(* PLC project mtcs_axes, Institute of Astronomy Onto 0.0.1 *)
(* stored: creationDateTime 2025-02-15T22:09:55.843531, modificationDateTime 2025-02-15T22:09:55.843531 *)

TYPE AxesIds : (AZI := 0, ABL := 1, ELE := 2, ROC := 3, RON := 4);
END_TYPE

TYPE AxesMoveUnits : (DEGREES := 0, RADIANS := 1, ARCSECONDS := 2);
END_TYPE

TYPE AxesAlphaUnits : (HOURS := 0, DEGREES := 1, RADIANS := 2);
END_TYPE

TYPE AxesDeltaUnits : (DEGREES := 0, RADIANS := 1);
END_TYPE

TYPE AxesMuUnits : (ARCSECONDS_PER_YEAR := 0, MILLIARCSECONDS_PER_YEAR := 1, DEGREES_PER_YEAR := 2, RADIANS_PER_YEAR := 3);
END_TYPE

TYPE AxesMoveVelocityUnits : (DEGREES_PER_SECOND := 0, ARCSECONDS_PER_SECOND := 1, RADIANS_PER_SECOND := 2, ARCSECONDS_PER_MINUTE := 3, ARCSECONDS_PER_HOUR := 4);
END_TYPE

TYPE AxesRotatorActivity : (NONE_ACTIVE := 0, ROC_ACTIVE := 1, RON_ACTIVE := 2);
END_TYPE

TYPE AxesParts : STRUCT
  {attribute 'TcHmiSymbol.Show'}
  azi : AxesAzimuthAxis;  (* The azimuth axis *)
  {attribute 'TcHmiSymbol.Show'}
  ele : AxesElevationAxis;  (* The elevation axis *)
  {attribute 'TcHmiSymbol.Show'}
  roc : AxesRotationAxis;  (* The cassegrain derotator axis *)
  {attribute 'TcHmiSymbol.Show'}
  ron : AxesRotationAxis;  (* The nasmyth derotator axis *)
  {attribute 'TcHmiSymbol.Show'}
  io : AxesIO;  (* I/O modules and drives *)
  {attribute 'TcHmiSymbol.Show'}
  configManager : ConfigManager;  (* The config manager (to load/save/activate configuration data) *)
  {attribute 'TcHmiSymbol.Show'}
  tpoint : AxesPointingModelsSetup;  (* The TPOINT models setup *)
END_STRUCT;
END_TYPE

TYPE AxesAzimuthAxisParts : STRUCT
  {attribute 'TcHmiSymbol.Show'}
  virtualAxis : AngularAxis;  (* The virtual AZI axis *)
  {attribute 'TcHmiSymbol.Show'}
  physicalAxis : AngularAxis;  (* The physical AZI axis *)
  {attribute 'TcHmiSymbol.Show'}
  ablAxis : AngularAxis;  (* The (anti-backlash) ABL axis *)
  {attribute 'TcHmiSymbol.Show'}
  lida1 : IncrementalEncoder;  (* The external (LIDA) encoder no. 1 *)
  {attribute 'TcHmiSymbol.Show'}
  lida2 : IncrementalEncoder;  (* The external (LIDA) encoder no. 2 *)
  {attribute 'TcHmiSymbol.Show'}
  lida3 : IncrementalEncoder;  (* The external (LIDA) encoder no. 3 *)
  {attribute 'TcHmiSymbol.Show'}
  lida4 : IncrementalEncoder;  (* The external (LIDA) encoder no. 4 *)
  {attribute 'TcHmiSymbol.Show'}
  absoluteEncoder : SSIEncoder;  (* The external absolute encoder *)
END_STRUCT;
END_TYPE

TYPE AxesElevationAxisParts : STRUCT
  {attribute 'TcHmiSymbol.Show'}
  virtualAxis : AngularAxis;  (* The virtual axis *)
  {attribute 'TcHmiSymbol.Show'}
  physicalAxis : AngularAxis;  (* The physical ELE axis *)
  {attribute 'TcHmiSymbol.Show'}
  lida1 : IncrementalEncoder;  (* The external (LIDA) encoder no. 1 *)
  {attribute 'TcHmiSymbol.Show'}
  lida2 : IncrementalEncoder;  (* The external (LIDA) encoder no. 2 *)
  {attribute 'TcHmiSymbol.Show'}
  absoluteEncoder : SSIEncoder;  (* The external absolute encoder *)
END_STRUCT;
END_TYPE

TYPE AxesRotationAxisParts : STRUCT
  {attribute 'TcHmiSymbol.Show'}
  virtualAxis : AngularAxis;  (* The virtual axis *)
  {attribute 'TcHmiSymbol.Show'}
  physicalAxis : AngularAxis;  (* The physical axis *)
END_STRUCT;
END_TYPE

TYPE AxesPointingModelSetupParts : STRUCT
  {attribute 'TcHmiSymbol.Show'}
  configManager : ConfigManager;  (* The config manager (to load/save/activate configuration data) *)
END_STRUCT;
END_TYPE

TYPE AxesPointingModelsSetupParts : STRUCT
  {attribute 'TcHmiSymbol.Show'}
  model0 : AxesPointingModelSetup;
  {attribute 'TcHmiSymbol.Show'}
  model1 : AxesPointingModelSetup;
  {attribute 'TcHmiSymbol.Show'}
  model2 : AxesPointingModelSetup;
  {attribute 'TcHmiSymbol.Show'}
  model3 : AxesPointingModelSetup;
  {attribute 'TcHmiSymbol.Show'}
  model4 : AxesPointingModelSetup;
  {attribute 'TcHmiSymbol.Show'}
  model5 : AxesPointingModelSetup;
  {attribute 'TcHmiSymbol.Show'}
  model6 : AxesPointingModelSetup;
  {attribute 'TcHmiSymbol.Show'}
  model7 : AxesPointingModelSetup;
  {attribute 'TcHmiSymbol.Show'}
  model8 : AxesPointingModelSetup;
  {attribute 'TcHmiSymbol.Show'}
  model9 : AxesPointingModelSetup;
END_STRUCT;
END_TYPE

TYPE AxesIOParts : STRUCT
  {attribute 'TcHmiSymbol.Show'}
  aziDrive : AX52XXDrive;  (* The AX5000 drive for the AZI en ROC motors *)
  {attribute 'TcHmiSymbol.Show'}
  ablDrive : AX52XXDrive;  (* The AX5000 drive for the ABL en RON motors *)
  {attribute 'TcHmiSymbol.Show'}
  eleDrive : AX52XXDrive;  (* The AX5000 drive for the ELE en FW motors *)
  {attribute 'TcHmiSymbol.Show'}
  TA_AZID : EtherCatDevice;  (* Telescope Axis - AZID *)
  {attribute 'TcHmiSymbol.Show'}
  TA_ABLD : EtherCatDevice;  (* Telescope Axis - ABLD *)
  {attribute 'TcHmiSymbol.Show'}
  TA_ELED : EtherCatDevice;  (* Telescope Axis - ELED *)
  {attribute 'TcHmiSymbol.Show'}
  TE_COU : EtherCatDevice;  (* Telescope Encoders - COU *)
  {attribute 'TcHmiSymbol.Show'}
  TE_EN1 : EtherCatDevice;  (* Telescope Encoders - EN1 *)
  {attribute 'TcHmiSymbol.Show'}
  TE_EN2 : EtherCatDevice;  (* Telescope Encoders - EN2 *)
  {attribute 'TcHmiSymbol.Show'}
  TE_EN3 : EtherCatDevice;  (* Telescope Encoders - EN3 *)
  {attribute 'TcHmiSymbol.Show'}
  TE_EN4 : EtherCatDevice;  (* Telescope Encoders - EN4 *)
  {attribute 'TcHmiSymbol.Show'}
  TE_EN5 : EtherCatDevice;  (* Telescope Encoders - EN5 *)
  {attribute 'TcHmiSymbol.Show'}
  TE_EN6 : EtherCatDevice;  (* Telescope Encoders - EN6 *)
  {attribute 'TcHmiSymbol.Show'}
  TE_EN7 : EtherCatDevice;  (* Telescope Encoders - EN7 *)
END_STRUCT;
END_TYPE

TYPE AxesProcesses : STRUCT
  {attribute 'TcHmiSymbol.Show'}
  initialize : Process;  (* Start initializing *)
  {attribute 'TcHmiSymbol.Show'}
  reset : Process;  (* Reset the axis (no homing) *)
  {attribute 'TcHmiSymbol.Show'}
  lock : Process;  (* Lock the system *)
  {attribute 'TcHmiSymbol.Show'}
  unlock : Process;  (* Unlock the system *)
  {attribute 'TcHmiSymbol.Show'}
  changeOperatingState : ChangeOperatingStateProcess;  (* Change the operating state (e.g. AUTO, MANUAL, ...) *)
  {attribute 'TcHmiSymbol.Show'}
  setTarget : AxesSetTargetProcess;  (* Set a new target *)
  {attribute 'TcHmiSymbol.Show'}
  point : AxesPointProcess;  (* Point the telescope to a new target *)
  {attribute 'TcHmiSymbol.Show'}
  pointRelative : AxesPointRelativeProcess;  (* Point the telescope relative to the current target *)
  {attribute 'TcHmiSymbol.Show'}
  stop : AxesStopProcess;  (* Stop the axes (i.e. stop pointing, tracking, moving, ...) *)
  {attribute 'TcHmiSymbol.Show'}
  quickStop : AxesStopProcess;  (* Quickly stop the axes (i.e. stop pointing, tracking, moving, ...) *)
  {attribute 'TcHmiSymbol.Show'}
  powerOn : AxesMultiPowerOnProcess;  (* Power on the axes *)
  {attribute 'TcHmiSymbol.Show'}
  powerOff : AxesPowerOffProcess;  (* Power off the axes *)
  {attribute 'TcHmiSymbol.Show'}
  doHoming : AxesDoHomingProcess;  (* Do a homing of the axes *)
  {attribute 'TcHmiSymbol.Show'}
  moveAbsolute : AxesMultiMoveProcess;  (* Move the axes in alt-azimuth to an absolute position *)
  {attribute 'TcHmiSymbol.Show'}
  moveRelative : AxesMultiMoveProcess;  (* Move the axes in alt-azimuth relative to the current position *)
  {attribute 'TcHmiSymbol.Show'}
  moveKnownPosition : AxesMoveKnownPositionProcess;  (* Move the axes to the given known position *)
  {attribute 'TcHmiSymbol.Show'}
  enablePointingModel : AxesEnablePointingModelProcess;  (* Enable a pointing model with the given name *)
  {attribute 'TcHmiSymbol.Show'}
  disablePointingModel : Process;  (* Disable the currently active pointing model *)
  {attribute 'TcHmiSymbol.Show'}
  setAlphaDeltaVelocity : AxesSetAlphaDeltaVelocityProcess;  (* Set an additional alpha/delta velocity (e.g. to track solar system objects) *)
END_STRUCT;
END_TYPE

TYPE AxesAzimuthAxisProcesses : STRUCT
  {attribute 'TcHmiSymbol.Show'}
  moveAbsolute : AxesMoveAbsoluteProcess;  (* Move the axis in an absolute way *)
  {attribute 'TcHmiSymbol.Show'}
  moveRelative : AxesMoveRelativeProcess;  (* Move the axis relative to the current position *)
  {attribute 'TcHmiSymbol.Show'}
  moveVelocity : AxesMoveVelocityProcess;  (* Move the axis endlessly with the given velocity *)
  {attribute 'TcHmiSymbol.Show'}
  reset : Process;  (* Reset the axis (no homing) *)
  {attribute 'TcHmiSymbol.Show'}
  moveOutOfLimitSwitch : AxesMoveOutOfLimitSwitchProcess;  (* Move out of a limit switch *)
  {attribute 'TcHmiSymbol.Show'}
  powerOn : AxesPowerOnProcess;  (* Power on the axis *)
  {attribute 'TcHmiSymbol.Show'}
  powerOff : AxesPowerOffProcess;  (* Power off the axis *)
  {attribute 'TcHmiSymbol.Show'}
  doHoming : AxesDoHomingProcess;  (* Do a homing of the axis *)
  {attribute 'TcHmiSymbol.Show'}
  stop : AxesStopProcess;  (* Stop the axis (i.e. stop pointing, tracking, moving, ...) *)
  {attribute 'TcHmiSymbol.Show'}
  quickStop : AxesStopProcess;  (* Quickly stop the axes (i.e. stop pointing, tracking, moving, ...) *)
  {attribute 'TcHmiSymbol.Show'}
  unlockBrake : AxesUnlockBrakeProcess;  (* Temporarily unlock the brake *)
  {attribute 'TcHmiSymbol.Show'}
  setPosition : AxesSetPositionProcess;  (* Set the axis to the given position *)
END_STRUCT;
END_TYPE

TYPE AxesElevationAxisProcesses : STRUCT
  {attribute 'TcHmiSymbol.Show'}
  moveAbsolute : AxesMoveAbsoluteProcess;  (* Move the axis in an absolute way *)
  {attribute 'TcHmiSymbol.Show'}
  moveRelative : AxesMoveRelativeProcess;  (* Move the axis relative to the current position *)
  {attribute 'TcHmiSymbol.Show'}
  moveVelocity : AxesMoveVelocityProcess;  (* Move the axis endlessly with the given velocity *)
  {attribute 'TcHmiSymbol.Show'}
  reset : Process;  (* Reset the axis (no homing) *)
  {attribute 'TcHmiSymbol.Show'}
  moveOutOfLimitSwitch : AxesMoveOutOfLimitSwitchProcess;  (* Move out of a limit switch *)
  {attribute 'TcHmiSymbol.Show'}
  powerOn : AxesPowerOnProcess;  (* Power on the axis *)
  {attribute 'TcHmiSymbol.Show'}
  powerOff : AxesPowerOffProcess;  (* Power off the axis *)
  {attribute 'TcHmiSymbol.Show'}
  doHoming : AxesDoHomingProcess;  (* Do a homing of the axis *)
  {attribute 'TcHmiSymbol.Show'}
  stop : AxesStopProcess;  (* Stop the axis (i.e. stop pointing, tracking, moving, ...) *)
  {attribute 'TcHmiSymbol.Show'}
  quickStop : AxesStopProcess;  (* Quickly stop the axes (i.e. stop pointing, tracking, moving, ...) *)
  {attribute 'TcHmiSymbol.Show'}
  setPosition : AxesSetPositionProcess;  (* Set the axis to the given position *)
  {attribute 'TcHmiSymbol.Show'}
  unlockBrake : AxesUnlockBrakeProcess;  (* Temporarily unlock the brake *)
END_STRUCT;
END_TYPE

TYPE AxesRotationAxisProcesses : STRUCT
  {attribute 'TcHmiSymbol.Show'}
  moveAbsolute : AxesMoveAbsoluteProcess;  (* Move the axis in an absolute way *)
  {attribute 'TcHmiSymbol.Show'}
  moveRelative : AxesMoveRelativeProcess;  (* Move the axis relative to the current position *)
  {attribute 'TcHmiSymbol.Show'}
  moveVelocity : AxesMoveVelocityProcess;  (* Move the axis endlessly with the given velocity *)
  {attribute 'TcHmiSymbol.Show'}
  reset : Process;  (* Reset the axis (no homing) *)
  {attribute 'TcHmiSymbol.Show'}
  moveOutOfLimitSwitch : AxesMoveOutOfLimitSwitchProcess;  (* Move out of a limit switch *)
  {attribute 'TcHmiSymbol.Show'}
  powerOn : AxesPowerOnProcess;  (* Power on the axis *)
  {attribute 'TcHmiSymbol.Show'}
  powerOff : AxesPowerOffProcess;  (* Power off the axis *)
  {attribute 'TcHmiSymbol.Show'}
  stop : AxesStopProcess;  (* Stop the axis (i.e. stop pointing, tracking, moving, ...) *)
  {attribute 'TcHmiSymbol.Show'}
  quickStop : AxesStopProcess;  (* Quickly stop the axes (i.e. stop pointing, tracking, moving, ...) *)
  {attribute 'TcHmiSymbol.Show'}
  setPosition : AxesSetPositionProcess;  (* Set the axis to the given position *)
END_STRUCT;
END_TYPE

TYPE AxesStatuses : STRUCT
  {attribute 'TcHmiSymbol.Show'}
  initializationStatus : InitializationStatus;
  {attribute 'TcHmiSymbol.Show'}
  healthStatus : HealthStatus;
  {attribute 'TcHmiSymbol.Show'}
  busyStatus : BusyStatus;
  {attribute 'TcHmiSymbol.Show'}
  operatingStatus : OperatingStatus;
  {attribute 'TcHmiSymbol.Show'}
  poweredStatus : PoweredStatus;
END_STRUCT;
END_TYPE

TYPE AxesTargetStatuses : STRUCT
  {attribute 'TcHmiSymbol.Show'}
  healthStatus : HealthStatus;
END_STRUCT;
END_TYPE

TYPE AxesFeedbackStatuses : STRUCT
  {attribute 'TcHmiSymbol.Show'}
  healthStatus : HealthStatus;
END_STRUCT;
END_TYPE

TYPE AxesAzimuthAxisStatuses : STRUCT
  {attribute 'TcHmiSymbol.Show'}
  busyStatus : BusyStatus;  (* Is the axis in a busy state? *)
  {attribute 'TcHmiSymbol.Show'}
  healthStatus : HealthStatus;  (* Is the axis in a healthy state? *)
  {attribute 'TcHmiSymbol.Show'}
  poweredStatus : PoweredStatus;  (* Is the axis powered on or off? *)
END_STRUCT;
END_TYPE

TYPE AxesElevationAxisStatuses : STRUCT
  {attribute 'TcHmiSymbol.Show'}
  busyStatus : BusyStatus;  (* Is the axis in a busy state? *)
  {attribute 'TcHmiSymbol.Show'}
  healthStatus : HealthStatus;  (* Is the axis in a healthy state? *)
  {attribute 'TcHmiSymbol.Show'}
  poweredStatus : PoweredStatus;  (* Is the axis powered on or off? *)
END_STRUCT;
END_TYPE

TYPE AxesRotationAxisStatuses : STRUCT
  {attribute 'TcHmiSymbol.Show'}
  busyStatus : BusyStatus;  (* Is the axis in a busy state? *)
  {attribute 'TcHmiSymbol.Show'}
  healthStatus : HealthStatus;  (* Is the axis in a healthy state? *)
  {attribute 'TcHmiSymbol.Show'}
  poweredStatus : PoweredStatus;  (* Is the axis powered on or off? *)
END_STRUCT;
END_TYPE

TYPE AxesPointingModelsSetupStatuses : STRUCT
  {attribute 'TcHmiSymbol.Show'}
  busyStatus : BusyStatus;  (* Is the pointing models setup in a busy state? *)
  {attribute 'TcHmiSymbol.Show'}
  healthStatus : HealthStatus;  (* Is the pointing models setup in a healthy state? *)
END_STRUCT;
END_TYPE

TYPE AxesIOStatuses : STRUCT
  {attribute 'TcHmiSymbol.Show'}
  healthStatus : HealthStatus;  (* Is the I/O in a healthy state? *)
END_STRUCT;
END_TYPE

TYPE AxesLocationConfig : STRUCT
  {attribute 'TcHmiSymbol.Show'}
  longitude : LREAL;  (* Observatory location: longitude [degrees, positive = E, negative = W] *)
  {attribute 'TcHmiSymbol.Show'}
  latitude : LREAL;  (* Observatory location: latitude [degrees, positive = N, negative = S] *)
  {attribute 'TcHmiSymbol.Show'}
  height : REAL;  (* Observatory location: height above sea-level [m] *)
  {attribute 'TcHmiSymbol.Show'}
  polarMotionX : REAL;  (* Earth polar motion x in degrees *)
  {attribute 'TcHmiSymbol.Show'}
  polarMotionY : REAL;  (* Earth polar motion y in degrees *)
  {attribute 'TcHmiSymbol.Show'}
  nutationDx : REAL;  (* Nutation adjustment dX in degrees *)
  {attribute 'TcHmiSymbol.Show'}
  nutationDy : REAL;  (* Nutation adjustment dY in degrees *)
END_STRUCT;
END_TYPE

TYPE AxesLocalConditionsConfig : STRUCT
  {attribute 'TcHmiSymbol.Show'}
  useTemperatureFromSensors : BOOL;  (* True if the temperature from the sensors should be used, false to use the temperature from the config *)
  {attribute 'TcHmiSymbol.Show'}
  configuredTemperature : REAL;  (* Local temperature in degrees, fixed by config *)
  {attribute 'TcHmiSymbol.Show'}
  configuredPressure : REAL;  (* Local temperature in hectoPascal = millibar, fixed by config *)
  {attribute 'TcHmiSymbol.Show'}
  useRelativeHumidityFromSensors : BOOL;  (* True if the temperature from the sensors should be used, false to use the temperature from the config *)
  {attribute 'TcHmiSymbol.Show'}
  configuredRelativeHumidity : REAL;  (* Local relative humidity as a fraction (0...1), fixed by config *)
  {attribute 'TcHmiSymbol.Show'}
  configuredObservingWavelength : REAL;  (* Observing wavelength in microns, fixed by config *)
  {attribute 'TcHmiSymbol.Show'}
  troposphericLapseRate : REAL;  (* Tropospheric lapse rate in K/m *)
END_STRUCT;
END_TYPE

TYPE AxesAzimuthConfig : STRUCT
  {attribute 'TcHmiSymbol.Show'}
  absoluteEncoderOffset : LREAL;  (* Offset in degrees, of the absolute encoder, w.r.t. zero *)
  {attribute 'TcHmiSymbol.Show'}
  absoluteEncoderInvert : BOOL;  (* TRUE to invert the counting direction of the absolute encoder *)
  {attribute 'TcHmiSymbol.Show'}
  lidasInvert : BOOL;  (* TRUE to invert the counting direction of the LIDAs *)
  {attribute 'TcHmiSymbol.Show'}
  moveOutOfLimitSwitchDistance : LREAL;  (* How many degrees should the moveOutOfLimitSwitch process try to move? *)
  {attribute 'TcHmiSymbol.Show'}
  positiveLimitSwitchInput : SINT;  (* Which input (0-7) represents the positive limit switch? *)
  {attribute 'TcHmiSymbol.Show'}
  negativeLimitSwitchInput : SINT;  (* Which input (0-7) represents the negative limit switch? *)
  {attribute 'TcHmiSymbol.Show'}
  minPositionLimitVirtualAxis : LREAL;  (* Limit the minimum position of the virtual axis to this value in degrees *)
  {attribute 'TcHmiSymbol.Show'}
  maxPositionLimitVirtualAxis : LREAL;  (* Limit the maximum position of the virtual axis to this value in degrees *)
  {attribute 'TcHmiSymbol.Show'}
  minPositionLimitPhysicalAxis : LREAL;  (* Limit the minimum position of the physical axis to this value in degrees *)
  {attribute 'TcHmiSymbol.Show'}
  maxPositionLimitPhysicalAxis : LREAL;  (* Limit the maximum position of the physical axis to this value in degrees *)
  {attribute 'TcHmiSymbol.Show'}
  velocityLimit : LREAL;  (* Limit the velocity of the axis to this value in degrees/sec *)
  {attribute 'TcHmiSymbol.Show'}
  accelerationLimit : LREAL;  (* Limit the acceleration (or deceleration) of the axis to this value in degrees/sec^2 *)
  {attribute 'TcHmiSymbol.Show'}
  minPositionSetpoint : LREAL;  (* The minimum position setpoint of the axis in degrees (should be a bit before the minPositionLimit) *)
  {attribute 'TcHmiSymbol.Show'}
  maxPositionSetpoint : LREAL;  (* The maximum position setpoint of the axis in degrees (should be a bit before the maxPositionLimit) *)
  {attribute 'TcHmiSymbol.Show'}
  maxVelocitySetpoint : LREAL;  (* The maximum velocity setpoint of the axis in degrees/sec *)
  {attribute 'TcHmiSymbol.Show'}
  maxAccelerationSetpoint : LREAL;  (* The maximum acceleration setpoint of the axis in degrees/sec^2 *)
  {attribute 'TcHmiSymbol.Show'}
  slipLimit : LREAL;  (* If the difference between the LIDA-encoder and motor-encoder positions is above this value in degrees, then we have detected slip *)
  {attribute 'TcHmiSymbol.Show'}
  ablMaxTorqueRiseSpeed : LREAL;  (* The ABL torque can rise maximum ... Nm/s on the telescope axis (always >0) *)
  {attribute 'TcHmiSymbol.Show'}
  ablMaxTorqueFallSpeed : LREAL;  (* The ABL torque can fall maximum ... Nm/s on the telescope axis (always >0) *)
  {attribute 'TcHmiSymbol.Show'}
  ablMaxTorque : LREAL;  (* The maximum ABL torque in Nm/s on the telescope axis (always >0) *)
  {attribute 'TcHmiSymbol.Show'}
  ablMinTorque : LREAL;  (* The minimum ABL torque in Nm/s on the telescope axis (always >0) *)
  {attribute 'TcHmiSymbol.Show'}
  ablZeroAccTorque : LREAL;  (* The ABL torque when the axis is not accelerating or decelerating (always >0) *)
  {attribute 'TcHmiSymbol.Show'}
  ablTorqueOutputOverride : LREAL;  (* Scale the ABL output torque by this fraction value (only for testing purposes, must be 1 normally!) *)
  {attribute 'TcHmiSymbol.Show'}
  ablPositiveTorque : BOOL;  (* True if a positive torque must be applied, false if a negative torque must be applied *)
  {attribute 'TcHmiSymbol.Show'}
  aziAndAblSameDirection : BOOL;  (* True if the AZI and ABL axes rotate in the same direction? *)
  {attribute 'TcHmiSymbol.Show'}
  homingHomePosition : LREAL;  (* The position of the homing mark (in degrees), with respect to the absolute zero *)
  {attribute 'TcHmiSymbol.Show'}
  homingStartAbsEncPosition : LREAL;  (* Absolute encoder position where the homing should go to first, in degrees *)
  {attribute 'TcHmiSymbol.Show'}
  homingGotoStartVelocity : LREAL;  (* Velocity when going to the start position, in degrees/sec *)
  {attribute 'TcHmiSymbol.Show'}
  homingVelocity : LREAL;  (* Velocity to search for the homing mark, in degrees/sec *)
  {attribute 'TcHmiSymbol.Show'}
  homingRange : LREAL;  (* Maximum distance to be covered while searching for the homing mark, in degrees *)
  {attribute 'TcHmiSymbol.Show'}
  quickStopDeceleration : LREAL;  (* Quick stop deceleration, in degrees/sec2 *)
  {attribute 'TcHmiSymbol.Show'}
  quickStopJerk : LREAL;  (* Quick stop jerk, in degrees/sec3 *)
END_STRUCT;
END_TYPE

TYPE AxesElevationConfig : STRUCT
  {attribute 'TcHmiSymbol.Show'}
  absoluteEncoderOffset : LREAL;  (* Offset in degrees, of the absolute encoder, w.r.t. zero *)
  {attribute 'TcHmiSymbol.Show'}
  absoluteEncoderInvert : BOOL;  (* TRUE to invert the counting direction *)
  {attribute 'TcHmiSymbol.Show'}
  lidasInvert : BOOL;  (* TRUE to invert the counting direction of the LIDAs *)
  {attribute 'TcHmiSymbol.Show'}
  moveOutOfLimitSwitchDistance : LREAL;  (* How many degrees should the moveOutOfLimitSwitch process try to move? *)
  {attribute 'TcHmiSymbol.Show'}
  positiveLimitSwitchInput : SINT;  (* Which input (0-7) represents the positive limit switch? *)
  {attribute 'TcHmiSymbol.Show'}
  negativeLimitSwitchInput : SINT;  (* Which input (0-7) represents the negative limit switch? *)
  {attribute 'TcHmiSymbol.Show'}
  minPositionLimitVirtualAxis : LREAL;  (* Limit the minimum position of the axis to this value in degrees, of the virtual axis *)
  {attribute 'TcHmiSymbol.Show'}
  maxPositionLimitVirtualAxis : LREAL;  (* Limit the maximum position of the axis to this value in degrees, of the virtual axis *)
  {attribute 'TcHmiSymbol.Show'}
  minPositionLimitPhysicalAxis : LREAL;  (* Limit the minimum position of the axis to this value in degrees, of the physical axis *)
  {attribute 'TcHmiSymbol.Show'}
  maxPositionLimitPhysicalAxis : LREAL;  (* Limit the maximum position of the axis to this value in degrees, of the physical axis *)
  {attribute 'TcHmiSymbol.Show'}
  velocityLimit : LREAL;  (* Limit the velocity of the axis to this value in degrees/sec *)
  {attribute 'TcHmiSymbol.Show'}
  accelerationLimit : LREAL;  (* Limit the acceleration (or deceleration) of the axis to this value in degrees/sec^2 *)
  {attribute 'TcHmiSymbol.Show'}
  minPositionSetpoint : LREAL;  (* The minimum position setpoint of the axis in degrees *)
  {attribute 'TcHmiSymbol.Show'}
  maxPositionSetpoint : LREAL;  (* The maximum position setpoint of the axis in degrees *)
  {attribute 'TcHmiSymbol.Show'}
  maxVelocitySetpoint : LREAL;  (* The maximum velocity setpoint of the axis in degrees/sec *)
  {attribute 'TcHmiSymbol.Show'}
  maxAccelerationSetpoint : LREAL;  (* The maximum acceleration setpoint of the axis in degrees/sec^2 *)
  {attribute 'TcHmiSymbol.Show'}
  slipLimit : LREAL;  (* If the difference between the LIDA-encoder and motor-encoder positions is above this value in degrees, then we have detected slip *)
  {attribute 'TcHmiSymbol.Show'}
  homingHomePosition : LREAL;  (* The position of the homing mark (in degrees), with respect to the absolute zero *)
  {attribute 'TcHmiSymbol.Show'}
  homingStartAbsEncPosition : LREAL;  (* Absolute encoder position where the homing should go to first, in degrees *)
  {attribute 'TcHmiSymbol.Show'}
  homingGotoStartVelocity : LREAL;  (* Velocity when going to the start position, in degrees/sec *)
  {attribute 'TcHmiSymbol.Show'}
  homingVelocity : LREAL;  (* Velocity to search for the homing mark, in degrees/sec *)
  {attribute 'TcHmiSymbol.Show'}
  homingRange : LREAL;  (* Maximum distance to be covered while searching for the homing mark, in degrees *)
  {attribute 'TcHmiSymbol.Show'}
  quickStopDeceleration : LREAL;  (* Quick stop deceleration, in degrees/sec2 *)
  {attribute 'TcHmiSymbol.Show'}
  quickStopJerk : LREAL;  (* Quick stop jerk, in degrees/sec3 *)
END_STRUCT;
END_TYPE

TYPE AxesRotationConfig : STRUCT
  {attribute 'TcHmiSymbol.Show'}
  motorEncoderOffset : LREAL;  (* Offset in degrees, of the absolute motor encoder, w.r.t. zero *)
  {attribute 'TcHmiSymbol.Show'}
  moveOutOfLimitSwitchDistance : LREAL;  (* How many degrees should the moveOutOfLimitSwitch process try to move? *)
  {attribute 'TcHmiSymbol.Show'}
  positiveLimitSwitchInput : SINT;  (* Which input (0-7) represents the positive limit switch? *)
  {attribute 'TcHmiSymbol.Show'}
  negativeLimitSwitchInput : SINT;  (* Which input (0-7) represents the negative limit switch? *)
  {attribute 'TcHmiSymbol.Show'}
  minPositionLimitVirtualAxis : LREAL;  (* Limit the minimum position of the axis to this value in degrees, of the virtual axis *)
  {attribute 'TcHmiSymbol.Show'}
  maxPositionLimitVirtualAxis : LREAL;  (* Limit the maximum position of the axis to this value in degrees, of the virtual axis *)
  {attribute 'TcHmiSymbol.Show'}
  minPositionLimitPhysicalAxis : LREAL;  (* Limit the minimum position of the axis to this value in degrees, of the physical axis *)
  {attribute 'TcHmiSymbol.Show'}
  maxPositionLimitPhysicalAxis : LREAL;  (* Limit the maximum position of the axis to this value in degrees, of the physical axis *)
  {attribute 'TcHmiSymbol.Show'}
  velocityLimit : LREAL;  (* Limit the velocity of the axis to this value in degrees/sec *)
  {attribute 'TcHmiSymbol.Show'}
  accelerationLimit : LREAL;  (* Limit the acceleration (or deceleration) of the axis to this value in degrees/sec^2 *)
  {attribute 'TcHmiSymbol.Show'}
  minPositionSetpoint : LREAL;  (* The minimum position setpoint of the axis in degrees *)
  {attribute 'TcHmiSymbol.Show'}
  maxPositionSetpoint : LREAL;  (* The maximum position setpoint of the axis in degrees *)
  {attribute 'TcHmiSymbol.Show'}
  maxVelocitySetpoint : LREAL;  (* The maximum velocity setpoint of the axis in degrees/sec *)
  {attribute 'TcHmiSymbol.Show'}
  maxAccelerationSetpoint : LREAL;  (* The maximum acceleration setpoint of the axis in degrees/sec^2 *)
  {attribute 'TcHmiSymbol.Show'}
  quickStopDeceleration : LREAL;  (* Quick stop deceleration, in degrees/sec2 *)
  {attribute 'TcHmiSymbol.Show'}
  quickStopJerk : LREAL;  (* Quick stop jerk, in degrees/sec3 *)
END_STRUCT;
END_TYPE

TYPE AxesKnownPositionConfig : STRUCT
  {attribute 'TcHmiSymbol.Show'}
  name : STRING;  (* The name of the position (e.g. 'PARK') *)
  {attribute 'TcHmiSymbol.Show'}
  allowObserver : BOOL;  (* Can an observer switch to this position? *)
  {attribute 'TcHmiSymbol.Show'}
  azi : LREAL;  (* Azimuth in degrees *)
  {attribute 'TcHmiSymbol.Show'}
  ele : LREAL;  (* Elevation in degrees *)
  {attribute 'TcHmiSymbol.Show'}
  roc : LREAL;  (* Cassegrain rotation in degrees *)
  {attribute 'TcHmiSymbol.Show'}
  ron : LREAL;  (* Nasmyth B rotation in degrees *)
  {attribute 'TcHmiSymbol.Show'}
  doAzi : BOOL;  (* Change the azimuth axis to the 'azi' position *)
  {attribute 'TcHmiSymbol.Show'}
  doEle : BOOL;  (* Change the elevation axis to the 'ele' position *)
  {attribute 'TcHmiSymbol.Show'}
  doRoc : BOOL;  (* Change the cassegrain rotation axis to the 'roc' position *)
  {attribute 'TcHmiSymbol.Show'}
  doRon : BOOL;  (* Change the nasmyth rotation axis to the 'ron' position *)
END_STRUCT;
END_TYPE

TYPE AxesKnownPositionsConfig : STRUCT
  {attribute 'TcHmiSymbol.Show'}
  position0 : AxesKnownPositionConfig;  (* Known position 0 *)
  {attribute 'TcHmiSymbol.Show'}
  position1 : AxesKnownPositionConfig;  (* Known position 1 *)
  {attribute 'TcHmiSymbol.Show'}
  position2 : AxesKnownPositionConfig;  (* Known position 2 *)
  {attribute 'TcHmiSymbol.Show'}
  position3 : AxesKnownPositionConfig;  (* Known position 3 *)
  {attribute 'TcHmiSymbol.Show'}
  position4 : AxesKnownPositionConfig;  (* Known position 4 *)
  {attribute 'TcHmiSymbol.Show'}
  position5 : AxesKnownPositionConfig;  (* Known position 5 *)
  {attribute 'TcHmiSymbol.Show'}
  position6 : AxesKnownPositionConfig;  (* Known position 6 *)
  {attribute 'TcHmiSymbol.Show'}
  position7 : AxesKnownPositionConfig;  (* Known position 7 *)
  {attribute 'TcHmiSymbol.Show'}
  position8 : AxesKnownPositionConfig;  (* Known position 8 *)
  {attribute 'TcHmiSymbol.Show'}
  position9 : AxesKnownPositionConfig;  (* Known position 9 *)
  {attribute 'TcHmiSymbol.Show'}
  position10 : AxesKnownPositionConfig;  (* Known position 10 *)
  {attribute 'TcHmiSymbol.Show'}
  position11 : AxesKnownPositionConfig;  (* Known position 11 *)
  {attribute 'TcHmiSymbol.Show'}
  position12 : AxesKnownPositionConfig;  (* Known position 12 *)
  {attribute 'TcHmiSymbol.Show'}
  position13 : AxesKnownPositionConfig;  (* Known position 13 *)
  {attribute 'TcHmiSymbol.Show'}
  position14 : AxesKnownPositionConfig;  (* Known position 14 *)
  {attribute 'TcHmiSymbol.Show'}
  position15 : AxesKnownPositionConfig;  (* Known position 15 *)
  {attribute 'TcHmiSymbol.Show'}
  position16 : AxesKnownPositionConfig;  (* Known position 16 *)
  {attribute 'TcHmiSymbol.Show'}
  position17 : AxesKnownPositionConfig;  (* Known position 17 *)
  {attribute 'TcHmiSymbol.Show'}
  position18 : AxesKnownPositionConfig;  (* Known position 18 *)
  {attribute 'TcHmiSymbol.Show'}
  position19 : AxesKnownPositionConfig;  (* Known position 19 *)
END_STRUCT;
END_TYPE

TYPE AxesConfig : STRUCT
  {attribute 'TcHmiSymbol.Show'}
  location : AxesLocationConfig;  (* Location of the observatory *)
  {attribute 'TcHmiSymbol.Show'}
  localConditions : AxesLocalConditionsConfig;  (* Location of the observatory *)
  {attribute 'TcHmiSymbol.Show'}
  knownPositions : AxesKnownPositionsConfig;  (* Known (predefined) positions (e.g. could be Park, Cover, Park winter, Mirror washing, ...) *)
  {attribute 'TcHmiSymbol.Show'}
  azi : AxesAzimuthConfig;  (* Azimuth axis *)
  {attribute 'TcHmiSymbol.Show'}
  ele : AxesElevationConfig;  (* Elevation axis *)
  {attribute 'TcHmiSymbol.Show'}
  roc : AxesRotationConfig;  (* Cassegrain rotation axis *)
  {attribute 'TcHmiSymbol.Show'}
  ron : AxesRotationConfig;  (* Nasmyth rotation axis *)
  {attribute 'TcHmiSymbol.Show'}
  cassegrainRotatorName : STRING;  (* Name of the Cassegrain rotator *)
  {attribute 'TcHmiSymbol.Show'}
  nasmythRotatorName : STRING;  (* Name of the Nasmyth rotator *)
  {attribute 'TcHmiSymbol.Show'}
  rocGuiAngle : LREAL;  (* Amgle to show ROC in the GUI *)
  {attribute 'TcHmiSymbol.Show'}
  ronGuiAngle : LREAL;  (* Amgle to show RON in the GUI *)
  {attribute 'TcHmiSymbol.Show'}
  knownPositionToleranceAzi : LREAL;  (* Tolerance (in degrees) to determine if the telescope is at a known position in azi direction *)
  {attribute 'TcHmiSymbol.Show'}
  knownPositionToleranceEle : LREAL;  (* Tolerance (in degrees) to determine if the telescope is at a known position in ele direction *)
  {attribute 'TcHmiSymbol.Show'}
  knownPositionToleranceRoc : LREAL;  (* Tolerance (in degrees) to determine if the telescope is at a known position in roc direction *)
  {attribute 'TcHmiSymbol.Show'}
  knownPositionToleranceRon : LREAL;  (* Tolerance (in degrees) to determine if the telescope is at a known position in ron direction *)
  {attribute 'TcHmiSymbol.Show'}
  rocPositionAngleSign : INT;  (* -1 to invert the sign of the PA for the cas derotator, 1 for positive *)
  {attribute 'TcHmiSymbol.Show'}
  ronPositionAngleSign : INT;  (* -1 to invert the sign of the PA for the cas derotator, 1 for positive *)
  {attribute 'TcHmiSymbol.Show'}
  tpointAziSign : INT;  (* -1 or 1 to invert input for TPOINT: A *)
  {attribute 'TcHmiSymbol.Show'}
  tpointEleSign : INT;  (* -1 or 1 to invert input for TPOINT: E *)
  {attribute 'TcHmiSymbol.Show'}
  tpointDeltaAziSign : INT;  (* -1 or 1 to invert input for TPOINT: DA *)
  {attribute 'TcHmiSymbol.Show'}
  tpointDeltaEleSign : INT;  (* -1 or 1 to invert input for TPOINT: DE *)
  {attribute 'TcHmiSymbol.Show'}
  tpointOldFormulas : BOOL;  (* True to use the old formulas *)
  {attribute 'TcHmiSymbol.Show'}
  tpointConvertRawAlphaDelta : BOOL;  (* If True, raw encoder values will be converted to feedback.alpha and feedback.delta, instead of corrected encoder values. Only use for tech stuff! *)
END_STRUCT;
END_TYPE

TYPE AxesPointingModelConfig : STRUCT
  {attribute 'TcHmiSymbol.Show'}
  name : STRING;  (* This name can be matched against the instrument name in the MTCS config and the focal station name in the M3 config. *)
  {attribute 'TcHmiSymbol.Show'}
  IE : LREAL;  (* Index error in elevation *)
  {attribute 'TcHmiSymbol.Show'}
  IA : LREAL;  (* Index error in azimuth *)
  {attribute 'TcHmiSymbol.Show'}
  CA : LREAL;  (* Nonperpendicularity of elevation and pointing axes *)
  {attribute 'TcHmiSymbol.Show'}
  AN : LREAL;  (* NS misalignment of azimuth axis *)
  {attribute 'TcHmiSymbol.Show'}
  AW : LREAL;  (* EW misalignment of azimuth axis *)
  {attribute 'TcHmiSymbol.Show'}
  NPAE : LREAL;  (* Nonperpendicularity of azimuth and elevation axes *)
  {attribute 'TcHmiSymbol.Show'}
  NRX : LREAL;  (* Horizontal displacement of Nasmyth rotation *)
  {attribute 'TcHmiSymbol.Show'}
  NRY : LREAL;  (* Vertical displacement of Nasmyth rotation *)
  {attribute 'TcHmiSymbol.Show'}
  ACES : LREAL;  (* Az centering error (sin component) *)
  {attribute 'TcHmiSymbol.Show'}
  ACEC : LREAL;  (* Az centering error (cos component) *)
  {attribute 'TcHmiSymbol.Show'}
  ECES : LREAL;  (* El centering error (sin component) *)
  {attribute 'TcHmiSymbol.Show'}
  ECEC : LREAL;  (* El centering error (cos component) *)
  {attribute 'TcHmiSymbol.Show'}
  TF : LREAL;  (* Tube flexure - sin(zeta) law *)
  {attribute 'TcHmiSymbol.Show'}
  TX : LREAL;  (* Tube flexure - tan(zeta) law *)
  {attribute 'TcHmiSymbol.Show'}
  FLOP : LREAL;  (* Constant vertical displacement *)
  {attribute 'TcHmiSymbol.Show'}
  POX : LREAL;  (* The x-coordinate of a pointing origin on a derotator *)
  {attribute 'TcHmiSymbol.Show'}
  POY : LREAL;  (* The y-coordinate of a pointing origin on a derotator *)
END_STRUCT;
END_TYPE

TYPE AxesSetTargetProcessArgs : STRUCT
  {attribute 'TcHmiSymbol.Show'}
  alphaUnits : AxesAlphaUnits;  (* The units in which alpha is given *)
  {attribute 'TcHmiSymbol.Show'}
  alpha : LREAL;  (* Right ascention, in the units of the alphaUnits argument *)
  {attribute 'TcHmiSymbol.Show'}
  deltaUnits : AxesDeltaUnits;  (* The units in which delta is given *)
  {attribute 'TcHmiSymbol.Show'}
  delta : LREAL;  (* Declination, in the units of the deltaUnits argument *)
  {attribute 'TcHmiSymbol.Show'}
  muUnits : AxesMuUnits;  (* The units in which muAlpha and muDelta are given *)
  {attribute 'TcHmiSymbol.Show'}
  muAlpha : LREAL;  (* Right ascention proper motion, the units of muUmits (do not multiply by cos(delta)!) *)
  {attribute 'TcHmiSymbol.Show'}
  muDelta : LREAL;  (* Declination proper motion, in radians/year *)
  {attribute 'TcHmiSymbol.Show'}
  parallax : LREAL;  (* Object parallax, in arcseconds *)
  {attribute 'TcHmiSymbol.Show'}
  radialVelocity : LREAL;  (* Object radial velocity, in km/s *)
  {attribute 'TcHmiSymbol.Show'}
  epoch : LREAL := 2000.0;  (* Epoch, e.g. 2000.0 *)
END_STRUCT;
END_TYPE

TYPE AxesPointProcessArgs : STRUCT
  {attribute 'TcHmiSymbol.Show'}
  alphaUnits : AxesAlphaUnits;  (* The units in which alpha is given *)
  {attribute 'TcHmiSymbol.Show'}
  alpha : LREAL;  (* Right ascention, in the units of the alphaUnits argument *)
  {attribute 'TcHmiSymbol.Show'}
  deltaUnits : AxesDeltaUnits;  (* The units in which delta is given *)
  {attribute 'TcHmiSymbol.Show'}
  delta : LREAL;  (* Declination, in the units of the deltaUnits argument *)
  {attribute 'TcHmiSymbol.Show'}
  muUnits : AxesMuUnits;  (* The units in which muAlpha and muDelta are given *)
  {attribute 'TcHmiSymbol.Show'}
  muAlpha : LREAL;  (* Right ascention proper motion, the units of muUmits (do not multiply by cos(delta)!) *)
  {attribute 'TcHmiSymbol.Show'}
  muDelta : LREAL;  (* Declination proper motion, in radians/year *)
  {attribute 'TcHmiSymbol.Show'}
  parallax : LREAL;  (* Object parallax, in arcseconds *)
  {attribute 'TcHmiSymbol.Show'}
  radialVelocity : LREAL;  (* Object radial velocity, in km/s *)
  {attribute 'TcHmiSymbol.Show'}
  epoch : LREAL := 2000.0;  (* Epoch, e.g. 2000.0 *)
  {attribute 'TcHmiSymbol.Show'}
  tracking : BOOL := TRUE;  (* True to start tracking the object, false to Only do a pointing *)
  {attribute 'TcHmiSymbol.Show'}
  rotUnits : AxesMoveUnits;  (* Units of the 'rot', 'roc' and 'ron' arguments (RADIANS, DEGREES, ARCSECONDS, ...) *)
  {attribute 'TcHmiSymbol.Show'}
  rotOffset : LREAL;  (* Offset to move the currently active rotator (incompatible with 'roc' and 'ron' args) *)
  {attribute 'TcHmiSymbol.Show'}
  rocOffset : LREAL;  (* Offset to move the cassegrain rotation axis (incompatible with 'rot' arg) *)
  {attribute 'TcHmiSymbol.Show'}
  ronOffset : LREAL;  (* Offset to move the nasmyth rotation axis (incompatible with 'rot' arg) *)
  {attribute 'TcHmiSymbol.Show'}
  doRotOffset : BOOL;  (* True to move the currently active rotator, false to leave it untouched *)
  {attribute 'TcHmiSymbol.Show'}
  doRocOffset : BOOL;  (* True to move the cassegrain rotation axis, false to leave it untouched *)
  {attribute 'TcHmiSymbol.Show'}
  doRonOffset : BOOL;  (* True to move the nasmyth rotation axis, false to leave it untouched *)
END_STRUCT;
END_TYPE

TYPE AxesPointRelativeProcessArgs : STRUCT
  {attribute 'TcHmiSymbol.Show'}
  alphaUnits : AxesAlphaUnits;  (* The units in which alpha is given *)
  {attribute 'TcHmiSymbol.Show'}
  alpha : LREAL;  (* Right ascention, in the units of the alphaUnits argument *)
  {attribute 'TcHmiSymbol.Show'}
  deltaUnits : AxesDeltaUnits;  (* The units in which delta is given *)
  {attribute 'TcHmiSymbol.Show'}
  delta : LREAL;  (* Declination, in the units of the deltaUnits argument *)
END_STRUCT;
END_TYPE

TYPE AxesMoveRelativeProcessArgs : STRUCT
  {attribute 'TcHmiSymbol.Show'}
  units : AxesMoveUnits;  (* Units of the 'value' argument (RADIANS, DEGREES, ARCSECONDS, ...) *)
  {attribute 'TcHmiSymbol.Show'}
  value : LREAL;  (* Move the axis with this value (which units depends on the 'units' argument) *)
END_STRUCT;
END_TYPE

TYPE AxesMoveAbsoluteProcessArgs : STRUCT
  {attribute 'TcHmiSymbol.Show'}
  units : AxesMoveUnits;  (* Units of the 'value' argument (RADIANS, DEGREES, ARCSECONDS, ...) *)
  {attribute 'TcHmiSymbol.Show'}
  value : LREAL;  (* Move the axis to this value (which units depends on the 'units' argument) + the optional offset *)
  {attribute 'TcHmiSymbol.Show'}
  offset : LREAL;  (* Optional extra offset (which will not be added to the 'startPos' *)
END_STRUCT;
END_TYPE

TYPE AxesMoveKnownPositionProcessArgs : STRUCT
  {attribute 'TcHmiSymbol.Show'}
  name : STRING;  (* Name of the position to move to *)
END_STRUCT;
END_TYPE

TYPE AxesMoveVelocityProcessArgs : STRUCT
  {attribute 'TcHmiSymbol.Show'}
  units : AxesMoveVelocityUnits;  (* Units of the 'value' argument (RADIANS_PER_SECOND, DEGREES_PER_SECOND, ...) *)
  {attribute 'TcHmiSymbol.Show'}
  value : LREAL;  (* Move the axis with this velocity (which units depends on the 'units' argument) *)
END_STRUCT;
END_TYPE

TYPE AxesMoveOutOfLimitSwitchProcessArgs : STRUCT
  {attribute 'TcHmiSymbol.Show'}
  switch : LimitSwitches;  (* Positive or negative limit switch *)
END_STRUCT;
END_TYPE

TYPE AxesMultiPowerOnProcessArgs : STRUCT
  {attribute 'TcHmiSymbol.Show'}
  azi : BOOL;  (* TRUE to power on AZI *)
  {attribute 'TcHmiSymbol.Show'}
  ele : BOOL;  (* TRUE to power on ELE *)
  {attribute 'TcHmiSymbol.Show'}
  roc : BOOL;  (* TRUE to power on ROC *)
  {attribute 'TcHmiSymbol.Show'}
  ron : BOOL;  (* TRUE to power on RON *)
  {attribute 'TcHmiSymbol.Show'}
  fw : BOOL;  (* TRUE to power on FW *)
END_STRUCT;
END_TYPE

TYPE AxesSetAlphaDeltaVelocityProcessArgs : STRUCT
  {attribute 'TcHmiSymbol.Show'}
  units : AxesMoveVelocityUnits;  (* Units of the alphaVelocity and deltaVelocity *)
  {attribute 'TcHmiSymbol.Show'}
  alphaVelocity : LREAL;  (* Velocity in alpha direction *)
  {attribute 'TcHmiSymbol.Show'}
  deltaVelocity : LREAL;  (* Velocity in delta direction *)
END_STRUCT;
END_TYPE

TYPE AxesMultiMoveProcessArgs : STRUCT
  {attribute 'TcHmiSymbol.Show'}
  units : AxesMoveUnits;  (* Units of the 'azi', 'ele', 'roc' and 'ron' arguments (RADIANS, DEGREES, ARCSECONDS, ...) *)
  {attribute 'TcHmiSymbol.Show'}
  azi : LREAL;  (* Angle to move the azimuth axis *)
  {attribute 'TcHmiSymbol.Show'}
  ele : LREAL;  (* Angle to move the elevation axis *)
  {attribute 'TcHmiSymbol.Show'}
  rot : LREAL;  (* Angle to move the currently active rotator (incompatible with 'roc' and 'ron' args) *)
  {attribute 'TcHmiSymbol.Show'}
  roc : LREAL;  (* Angle to move the cassegrain rotation axis (incompatible with 'rot' arg) *)
  {attribute 'TcHmiSymbol.Show'}
  ron : LREAL;  (* Angle to move the nasmyth rotation axis (incompatible with 'rot' arg) *)
  {attribute 'TcHmiSymbol.Show'}
  doAzi : BOOL;  (* True to move the azimuth axis, false to leave it untouched *)
  {attribute 'TcHmiSymbol.Show'}
  doEle : BOOL;  (* True to move the elevation axis, false to leave it untouched *)
  {attribute 'TcHmiSymbol.Show'}
  doRot : BOOL;  (* True to move the currently active rotator, false to leave it untouched *)
  {attribute 'TcHmiSymbol.Show'}
  doRoc : BOOL;  (* True to move the cassegrain rotation axis, false to leave it untouched *)
  {attribute 'TcHmiSymbol.Show'}
  doRon : BOOL;  (* True to move the nasmyth rotation axis, false to leave it untouched *)
  {attribute 'TcHmiSymbol.Show'}
  preferMostTravel : BOOL := FALSE;  (* Only in case of relative movement during tracking: If possible, go to the position where there is most travel (if the telescope is tracking). If false, it will go there the quickest way possible. *)
END_STRUCT;
END_TYPE

TYPE AxesEnablePointingModelProcessArgs : STRUCT
  {attribute 'TcHmiSymbol.Show'}
  name : STRING;  (* Name of the pointing model *)
END_STRUCT;
END_TYPE

TYPE AxesUnlockBrakeProcessArgs : STRUCT
  {attribute 'TcHmiSymbol.Show'}
  seconds : LREAL := 10.0;  (* Unlock the brake for this number of seconds (0 means forever) *)
END_STRUCT;
END_TYPE

TYPE AxesSetPositionProcessArgs : STRUCT
  {attribute 'TcHmiSymbol.Show'}
  value : LREAL;  (* New position to be taken over by the axis *)
END_STRUCT;
END_TYPE

FUNCTION_BLOCK SM_Axes
  VAR_INPUT
    {attribute 'TcHmiSymbol.Show'}
    {attribute 'OPC.UA.DA' := '1'}
    {attribute 'OPC.UA.DA.Access' := '1'}
    editableConfig : AxesConfig;  (* Editable configuration of the Axes subsystem *)
    {attribute 'TcHmiSymbol.Show'}
    {attribute 'OPC.UA.DA' := '1'}
    {attribute 'OPC.UA.DA.Access' := '1'}
    fromCppAxes AT %I* : TmcToPlcAxes;  (* Data from the C++ task *)
  END_VAR
  VAR_OUTPUT
    {attribute 'OPC.UA.DA' := '1'}
    {attribute 'OPC.UA.DA.Access' := '1'}
    {attribute 'TcHmiSymbol.Show'}
    actualStatus : STRING;  (* Current status description *)
    {attribute 'TcHmiSymbol.Show'}
    previousStatus : STRING;  (* Previous status description *)
    {attribute 'TcHmiSymbol.Show'}
    {attribute 'OPC.UA.DA' := '1'}
    {attribute 'OPC.UA.DA.Access' := '1'}
    isPoweredOffByPersonInDome : BOOL;  (* True if the axes are powered off due to a person entering the dome *)
    {attribute 'TcHmiSymbol.Show'}
    {attribute 'OPC.UA.DA' := '1'}
    {attribute 'OPC.UA.DA.Access' := '1'}
    isPointing : BOOL;  (* True if the telescope is pointing *)
    {attribute 'TcHmiSymbol.Show'}
    {attribute 'OPC.UA.DA' := '1'}
    {attribute 'OPC.UA.DA.Access' := '1'}
    isLimitsReached : BOOL;  (* True if a positiom limit is reached *)
    {attribute 'TcHmiSymbol.Show'}
    {attribute 'OPC.UA.DA' := '1'}
    {attribute 'OPC.UA.DA.Access' := '1'}
    isTracking : BOOL;  (* True if the telescope is tracking *)
    {attribute 'TcHmiSymbol.Show'}
    {attribute 'OPC.UA.DA' := '1'}
    {attribute 'OPC.UA.DA.Access' := '1'}
    isOffsetting : BOOL;  (* True if the telescope is offsetting (movin *)
    {attribute 'TcHmiSymbol.Show'}
    {attribute 'OPC.UA.DA' := '1'}
    {attribute 'OPC.UA.DA.Access' := '1'}
    isAtKnownPosition : BOOL;  (* True if the telescope is at a known position *)
    {attribute 'TcHmiSymbol.Show'}
    {attribute 'OPC.UA.DA' := '1'}
    {attribute 'OPC.UA.DA.Access' := '1'}
    isPointingModelActive : BOOL;  (* Is a pointing model currently active? *)
    {attribute 'TcHmiSymbol.Show'}
    {attribute 'OPC.UA.DA' := '1'}
    {attribute 'OPC.UA.DA.Access' := '1'}
    activeRotator : AxesRotatorActivity;  (* Which rotator is active? *)
    {attribute 'TcHmiSymbol.Show'}
    {attribute 'OPC.UA.DA' := '1'}
    {attribute 'OPC.UA.DA.Access' := '1'}
    actualKnownPositionName : STRING;  (* Name of the known position if isAtKnownPosition is True *)
    {attribute 'TcHmiSymbol.Show'}
    {attribute 'OPC.UA.DA' := '1'}
    {attribute 'OPC.UA.DA.Access' := '1'}
    config : AxesConfig;  (* Active configuration of the Axes subsystem *)
    {attribute 'TcHmiSymbol.Show'}
    {attribute 'OPC.UA.DA' := '1'}
    {attribute 'OPC.UA.DA.Access' := '1'}
    toCppAxes AT %Q* : TmcFromPlcAxes;  (* Data to the C++ task *)
    {attribute 'TcHmiSymbol.Show'}
    {attribute 'OPC.UA.DA' := '1'}
    {attribute 'OPC.UA.DA.Access' := '1'}
    activePointingModel : AxesPointingModelConfig;  (* Currently active TPoint model (if isPointingModelActive is TRUE) *)
    {attribute 'TcHmiSymbol.Show'}
    {attribute 'OPC.UA.DA' := '1'}
    {attribute 'OPC.UA.DA.Access' := '1'}
    activePointingModelNumber : INT;  (* Number of the currently active TPoint model (if isPointingModelActive is TRUE), -1 if no model is active *)
    {attribute 'TcHmiSymbol.Show'}
    {attribute 'OPC.UA.DA' := '1'}
    {attribute 'OPC.UA.DA.Access' := '1'}
    target : AxesTarget;  (* The actual target *)
    {attribute 'TcHmiSymbol.Show'}
    {attribute 'OPC.UA.DA' := '1'}
    {attribute 'OPC.UA.DA.Access' := '1'}
    feedback : AxesFeedback;  (* The actual feedback *)
    {attribute 'TcHmiSymbol.Show'}
    statuses : AxesStatuses;  (* Statuses of the state machine *)
    {attribute 'TcHmiSymbol.Show'}
    parts : AxesParts;  (* Parts of the state machine *)
    {attribute 'TcHmiSymbol.Show'}
    processes : AxesProcesses;  (* Processes of the state machine *)
  END_VAR
  VAR_IN_OUT
    {attribute 'TcHmiSymbol.Show'}
    {attribute 'OPC.UA.DA' := '0'}
    {attribute 'TcHmiSymbol.Hide'}
    timing : ServicesTiming;  (* Reference to the timing service *)
    {attribute 'TcHmiSymbol.Show'}
    {attribute 'OPC.UA.DA' := '0'}
    {attribute 'TcHmiSymbol.Hide'}
    motionBlocking : SafetyMotionBlocking;  (* Reference to the motion blocking safety *)
    {attribute 'TcHmiSymbol.Show'}
    {attribute 'OPC.UA.DA' := '0'}
    {attribute 'TcHmiSymbol.Hide'}
    domeAccess : SafetyDomeAccess;  (* Reference to the dome access safety *)
    {attribute 'TcHmiSymbol.Show'}
    {attribute 'OPC.UA.DA' := '0'}
    {attribute 'TcHmiSymbol.Hide'}
    operatorStatus : OperatorStatus;  (* Shared operator status *)
    {attribute 'TcHmiSymbol.Show'}
    {attribute 'OPC.UA.DA' := '0'}
    {attribute 'TcHmiSymbol.Hide'}
    activityStatus : ActivityStatus;  (* Shared activity status *)
    {attribute 'TcHmiSymbol.Show'}
    {attribute 'OPC.UA.DA' := '0'}
    {attribute 'TcHmiSymbol.Hide'}
    activeInstrument : InstrumentConfig;  (* Instrument config *if* isInstrumentActive is TRUE *)
    {attribute 'TcHmiSymbol.Show'}
    {attribute 'OPC.UA.DA' := '0'}
    {attribute 'TcHmiSymbol.Hide'}
    isInstrumentActive : BOOL;  (* Is an instrument currently active (i.e. is M3 static at a known position?) *)
  END_VAR
  VAR
    {attribute 'TcHmiSymbol.Show'}
    {attribute 'OPC.UA.DA' := '1'}
    {attribute 'OPC.UA.DA.Access' := '1'}
    fromCppAxes_ro : TmcToPlcAxes;
  END_VAR

            parts.azi(
    isEnabled := (NOT(statuses.initializationStatus.locked)) AND operatorStatus.tech,
    id := AxesIds.AZI,
    config := config.azi,
    aziDriveChannel := parts.io.parts.aziDrive.parts.channelA,
    ablDriveChannel := parts.io.parts.ablDrive.parts.channelA,
    aziMainDriveChannel := parts.io.parts.aziDrive.parts.channelA,
    ablMainDriveChannel := parts.io.parts.ablDrive.parts.channelA);
parts.ele(
    isEnabled := (NOT(statuses.initializationStatus.locked)) AND operatorStatus.tech,
    id := AxesIds.ELE,
    config := config.ele,
    driveChannel := parts.io.parts.eleDrive.parts.channelA,
    mainDriveChannel := parts.io.parts.eleDrive.parts.channelA);
parts.roc(
    isEnabled := (NOT(statuses.initializationStatus.locked)) AND operatorStatus.tech,
    id := AxesIds.ROC,
    config := config.roc,
    driveChannel := parts.io.parts.aziDrive.parts.channelB,
    mainDriveChannel := parts.io.parts.aziDrive.parts.channelA);
parts.ron(
    isEnabled := (NOT(statuses.initializationStatus.locked)) AND operatorStatus.tech,
    id := AxesIds.RON,
    config := config.ron,
    driveChannel := parts.io.parts.ablDrive.parts.channelB,
    mainDriveChannel := parts.io.parts.ablDrive.parts.channelA);
parts.io( isEnabled := operatorStatus.tech );
parts.configManager( isEnabled := operatorStatus.tech );
parts.tpoint( isEnabled := operatorStatus.tech );
statuses.initializationStatus();
statuses.healthStatus(
    isGood := feedback.statuses.healthStatus.isGood AND (target.statuses.healthStatus.isGood AND (parts.azi.statuses.healthStatus.isGood AND (parts.ele.statuses.healthStatus.isGood AND (parts.roc.statuses.healthStatus.isGood AND (parts.ron.statuses.healthStatus.isGood AND (parts.configManager.statuses.healthStatus.isGood AND (parts.tpoint.statuses.healthStatus.isGood AND (parts.io.statuses.healthStatus.isGood AND (processes.initialize.statuses.healthStatus.isGood AND (processes.reset.statuses.healthStatus.isGood AND (processes.lock.statuses.healthStatus.isGood AND (processes.unlock.statuses.healthStatus.isGood AND (processes.changeOperatingState.statuses.healthStatus.isGood AND (processes.setTarget.statuses.healthStatus.isGood AND (processes.point.statuses.healthStatus.isGood AND (processes.pointRelative.statuses.healthStatus.isGood AND (processes.stop.statuses.healthStatus.isGood AND (processes.quickStop.statuses.healthStatus.isGood AND (processes.powerOn.statuses.healthStatus.isGood AND (processes.powerOff.statuses.healthStatus.isGood AND (processes.doHoming.statuses.healthStatus.isGood AND (processes.moveAbsolute.statuses.healthStatus.isGood AND (processes.moveRelative.statuses.healthStatus.isGood AND (processes.moveKnownPosition.statuses.healthStatus.isGood AND (processes.enablePointingModel.statuses.healthStatus.isGood AND (processes.disablePointingModel.statuses.healthStatus.isGood AND processes.setAlphaDeltaVelocity.statuses.healthStatus.isGood)))))))))))))))))))))))))),
    hasWarning := feedback.statuses.healthStatus.hasWarning OR (target.statuses.healthStatus.hasWarning OR (parts.azi.statuses.healthStatus.hasWarning OR (parts.ele.statuses.healthStatus.hasWarning OR (parts.roc.statuses.healthStatus.hasWarning OR (parts.ron.statuses.healthStatus.hasWarning OR (parts.configManager.statuses.healthStatus.hasWarning OR (parts.tpoint.statuses.healthStatus.hasWarning OR (parts.io.statuses.healthStatus.hasWarning OR (processes.initialize.statuses.healthStatus.hasWarning OR (processes.reset.statuses.healthStatus.hasWarning OR (processes.lock.statuses.healthStatus.hasWarning OR (processes.unlock.statuses.healthStatus.hasWarning OR (processes.changeOperatingState.statuses.healthStatus.hasWarning OR (processes.setTarget.statuses.healthStatus.hasWarning OR (processes.point.statuses.healthStatus.hasWarning OR (processes.pointRelative.statuses.healthStatus.hasWarning OR (processes.stop.statuses.healthStatus.hasWarning OR (processes.quickStop.statuses.healthStatus.hasWarning OR (processes.powerOn.statuses.healthStatus.hasWarning OR (processes.powerOff.statuses.healthStatus.hasWarning OR (processes.doHoming.statuses.healthStatus.hasWarning OR (processes.moveAbsolute.statuses.healthStatus.hasWarning OR (processes.moveRelative.statuses.healthStatus.hasWarning OR (processes.moveKnownPosition.statuses.healthStatus.hasWarning OR (processes.enablePointingModel.statuses.healthStatus.hasWarning OR (processes.disablePointingModel.statuses.healthStatus.hasWarning OR processes.setAlphaDeltaVelocity.statuses.healthStatus.hasWarning)))))))))))))))))))))))))));
statuses.busyStatus( isBusy := parts.azi.statuses.busyStatus.busy OR (parts.ele.statuses.busyStatus.busy OR (parts.roc.statuses.busyStatus.busy OR (parts.ron.statuses.busyStatus.busy OR (parts.configManager.statuses.busyStatus.busy OR (parts.tpoint.statuses.busyStatus.busy OR (processes.initialize.statuses.busyStatus.busy OR (processes.reset.statuses.busyStatus.busy OR (processes.lock.statuses.busyStatus.busy OR (processes.unlock.statuses.busyStatus.busy OR (processes.changeOperatingState.statuses.busyStatus.busy OR (processes.setTarget.statuses.busyStatus.busy OR (processes.point.statuses.busyStatus.busy OR (processes.pointRelative.statuses.busyStatus.busy OR (processes.stop.statuses.busyStatus.busy OR (processes.quickStop.statuses.busyStatus.busy OR (processes.powerOn.statuses.busyStatus.busy OR (processes.powerOff.statuses.busyStatus.busy OR (processes.doHoming.statuses.busyStatus.busy OR (processes.moveAbsolute.statuses.busyStatus.busy OR (processes.moveRelative.statuses.busyStatus.busy OR (processes.moveKnownPosition.statuses.busyStatus.busy OR (processes.enablePointingModel.statuses.busyStatus.busy OR (processes.disablePointingModel.statuses.busyStatus.busy OR processes.setAlphaDeltaVelocity.statuses.busyStatus.busy))))))))))))))))))))))) );
statuses.operatingStatus( superState := statuses.initializationStatus.initialized );
statuses.poweredStatus();
processes.initialize( isEnabled := (NOT(statuses.initializationStatus.locked)) AND (statuses.initializationStatus.shutdown OR (statuses.initializationStatus.initializingFailed OR statuses.initializationStatus.initialized)) );
processes.reset( isEnabled := TRUE );
processes.lock( isEnabled := operatorStatus.tech );
processes.unlock( isEnabled := operatorStatus.tech AND statuses.initializationStatus.locked );
processes.changeOperatingState( isEnabled := statuses.busyStatus.idle AND (statuses.initializationStatus.initialized AND operatorStatus.tech) );
processes.setTarget( isEnabled := statuses.initializationStatus.initialized AND operatorStatus.tech );
processes.point( isEnabled := statuses.initializationStatus.initialized AND (statuses.busyStatus.idle AND statuses.poweredStatus.enabled) );
processes.pointRelative( isEnabled := statuses.initializationStatus.initialized AND (statuses.busyStatus.idle AND statuses.poweredStatus.enabled) );
processes.stop( isEnabled := statuses.initializationStatus.initialized );
processes.quickStop( isEnabled := statuses.initializationStatus.initialized );
processes.powerOn( isEnabled := (NOT(statuses.initializationStatus.locked)) AND (statuses.initializationStatus.initialized AND processes.powerOn.statuses.busyStatus.idle) );
processes.powerOff( isEnabled := statuses.initializationStatus.initialized AND processes.powerOff.statuses.busyStatus.idle );
processes.doHoming( isEnabled := operatorStatus.tech );
processes.moveAbsolute( isEnabled := statuses.initializationStatus.initialized AND (statuses.busyStatus.idle AND statuses.poweredStatus.enabled) );
processes.moveRelative( isEnabled := statuses.initializationStatus.initialized AND (statuses.busyStatus.idle AND statuses.poweredStatus.enabled) );
processes.moveKnownPosition( isEnabled := statuses.initializationStatus.initialized AND (statuses.busyStatus.idle AND statuses.poweredStatus.enabled) );
processes.enablePointingModel( isEnabled := statuses.busyStatus.idle );
processes.disablePointingModel( isEnabled := statuses.busyStatus.idle );
processes.setAlphaDeltaVelocity( isEnabled := statuses.initializationStatus.initialized AND statuses.busyStatus.idle );
fromCppAxes_ro := fromCppAxes;

          

{attribute 'TcRpcEnable' := '1'}
METHOD initialize : RequestResults
                  initialize := THIS^.processes.initialize.request();

                
END_METHOD

{attribute 'TcRpcEnable' := '1'}
METHOD reset : RequestResults
                  reset := THIS^.processes.reset.request();

                
END_METHOD

{attribute 'TcRpcEnable' := '1'}
METHOD lock : RequestResults
                  lock := THIS^.processes.lock.request();

                
END_METHOD

{attribute 'TcRpcEnable' := '1'}
METHOD unlock : RequestResults
                  unlock := THIS^.processes.unlock.request();

                
END_METHOD

{attribute 'TcRpcEnable' := '1'}
METHOD changeOperatingState : RequestResults
  VAR_INPUT
    {attribute 'TcHmiSymbol.Show'}
    state : OperatingStates;
  END_VAR
                  changeOperatingState := THIS^.processes.changeOperatingState.request( state := state );

                
END_METHOD

{attribute 'TcRpcEnable' := '1'}
METHOD setTarget : RequestResults
  VAR_INPUT
    {attribute 'TcHmiSymbol.Show'}
    alphaUnits : AxesAlphaUnits;
    {attribute 'TcHmiSymbol.Show'}
    alpha : LREAL;
    {attribute 'TcHmiSymbol.Show'}
    deltaUnits : AxesDeltaUnits;
    {attribute 'TcHmiSymbol.Show'}
    delta : LREAL;
    {attribute 'TcHmiSymbol.Show'}
    muUnits : AxesMuUnits;
    {attribute 'TcHmiSymbol.Show'}
    muAlpha : LREAL;
    {attribute 'TcHmiSymbol.Show'}
    muDelta : LREAL;
    {attribute 'TcHmiSymbol.Show'}
    parallax : LREAL;
    {attribute 'TcHmiSymbol.Show'}
    radialVelocity : LREAL;
    {attribute 'TcHmiSymbol.Show'}
    epoch : LREAL;
  END_VAR
                  setTarget := THIS^.processes.setTarget.request(
    alphaUnits := alphaUnits,
    alpha := alpha,
    deltaUnits := deltaUnits,
    delta := delta,
    muUnits := muUnits,
    muAlpha := muAlpha,
    muDelta := muDelta,
    parallax := parallax,
    radialVelocity := radialVelocity,
    epoch := epoch);

                
END_METHOD

{attribute 'TcRpcEnable' := '1'}
METHOD point : RequestResults
  VAR_INPUT
    {attribute 'TcHmiSymbol.Show'}
    alphaUnits : AxesAlphaUnits;
    {attribute 'TcHmiSymbol.Show'}
    alpha : LREAL;
    {attribute 'TcHmiSymbol.Show'}
    deltaUnits : AxesDeltaUnits;
    {attribute 'TcHmiSymbol.Show'}
    delta : LREAL;
    {attribute 'TcHmiSymbol.Show'}
    muUnits : AxesMuUnits;
    {attribute 'TcHmiSymbol.Show'}
    muAlpha : LREAL;
    {attribute 'TcHmiSymbol.Show'}
    muDelta : LREAL;
    {attribute 'TcHmiSymbol.Show'}
    parallax : LREAL;
    {attribute 'TcHmiSymbol.Show'}
    radialVelocity : LREAL;
    {attribute 'TcHmiSymbol.Show'}
    epoch : LREAL;
    {attribute 'TcHmiSymbol.Show'}
    tracking : BOOL;
    {attribute 'TcHmiSymbol.Show'}
    rotUnits : AxesMoveUnits;
    {attribute 'TcHmiSymbol.Show'}
    rotOffset : LREAL;
    {attribute 'TcHmiSymbol.Show'}
    rocOffset : LREAL;
    {attribute 'TcHmiSymbol.Show'}
    ronOffset : LREAL;
    {attribute 'TcHmiSymbol.Show'}
    doRotOffset : BOOL;
    {attribute 'TcHmiSymbol.Show'}
    doRocOffset : BOOL;
    {attribute 'TcHmiSymbol.Show'}
    doRonOffset : BOOL;
  END_VAR
                  point := THIS^.processes.point.request(
    alphaUnits := alphaUnits,
    alpha := alpha,
    deltaUnits := deltaUnits,
    delta := delta,
    muUnits := muUnits,
    muAlpha := muAlpha,
    muDelta := muDelta,
    parallax := parallax,
    radialVelocity := radialVelocity,
    epoch := epoch,
    tracking := tracking,
    rotUnits := rotUnits,
    rotOffset := rotOffset,
    rocOffset := rocOffset,
    ronOffset := ronOffset,
    doRotOffset := doRotOffset,
    doRocOffset := doRocOffset,
    doRonOffset := doRonOffset);

                
END_METHOD

{attribute 'TcRpcEnable' := '1'}
METHOD pointRelative : RequestResults
  VAR_INPUT
    {attribute 'TcHmiSymbol.Show'}
    alphaUnits : AxesAlphaUnits;
    {attribute 'TcHmiSymbol.Show'}
    alpha : LREAL;
    {attribute 'TcHmiSymbol.Show'}
    deltaUnits : AxesDeltaUnits;
    {attribute 'TcHmiSymbol.Show'}
    delta : LREAL;
  END_VAR
                  pointRelative := THIS^.processes.pointRelative.request(
    alphaUnits := alphaUnits,
    alpha := alpha,
    deltaUnits := deltaUnits,
    delta := delta);

                
END_METHOD

{attribute 'TcRpcEnable' := '1'}
METHOD stop : RequestResults
                  stop := THIS^.processes.stop.request();

                
END_METHOD

{attribute 'TcRpcEnable' := '1'}
METHOD quickStop : RequestResults
                  quickStop := THIS^.processes.quickStop.request();

                
END_METHOD

{attribute 'TcRpcEnable' := '1'}
METHOD powerOn : RequestResults
  VAR_INPUT
    {attribute 'TcHmiSymbol.Show'}
    azi : BOOL;
    {attribute 'TcHmiSymbol.Show'}
    ele : BOOL;
    {attribute 'TcHmiSymbol.Show'}
    roc : BOOL;
    {attribute 'TcHmiSymbol.Show'}
    ron : BOOL;
    {attribute 'TcHmiSymbol.Show'}
    fw : BOOL;
  END_VAR
                  powerOn := THIS^.processes.powerOn.request(
    azi := azi,
    ele := ele,
    roc := roc,
    ron := ron,
    fw := fw);

                
END_METHOD

{attribute 'TcRpcEnable' := '1'}
METHOD powerOff : RequestResults
                  powerOff := THIS^.processes.powerOff.request();

                
END_METHOD

{attribute 'TcRpcEnable' := '1'}
METHOD doHoming : RequestResults
                  doHoming := THIS^.processes.doHoming.request();

                
END_METHOD

{attribute 'TcRpcEnable' := '1'}
METHOD moveAbsolute : RequestResults
  VAR_INPUT
    {attribute 'TcHmiSymbol.Show'}
    units : AxesMoveUnits;
    {attribute 'TcHmiSymbol.Show'}
    azi : LREAL;
    {attribute 'TcHmiSymbol.Show'}
    ele : LREAL;
    {attribute 'TcHmiSymbol.Show'}
    rot : LREAL;
    {attribute 'TcHmiSymbol.Show'}
    roc : LREAL;
    {attribute 'TcHmiSymbol.Show'}
    ron : LREAL;
    {attribute 'TcHmiSymbol.Show'}
    doAzi : BOOL;
    {attribute 'TcHmiSymbol.Show'}
    doEle : BOOL;
    {attribute 'TcHmiSymbol.Show'}
    doRot : BOOL;
    {attribute 'TcHmiSymbol.Show'}
    doRoc : BOOL;
    {attribute 'TcHmiSymbol.Show'}
    doRon : BOOL;
    {attribute 'TcHmiSymbol.Show'}
    preferMostTravel : BOOL;
  END_VAR
                  moveAbsolute := THIS^.processes.moveAbsolute.request(
    units := units,
    azi := azi,
    ele := ele,
    rot := rot,
    roc := roc,
    ron := ron,
    doAzi := doAzi,
    doEle := doEle,
    doRot := doRot,
    doRoc := doRoc,
    doRon := doRon,
    preferMostTravel := preferMostTravel);

                
END_METHOD

{attribute 'TcRpcEnable' := '1'}
METHOD moveRelative : RequestResults
  VAR_INPUT
    {attribute 'TcHmiSymbol.Show'}
    units : AxesMoveUnits;
    {attribute 'TcHmiSymbol.Show'}
    azi : LREAL;
    {attribute 'TcHmiSymbol.Show'}
    ele : LREAL;
    {attribute 'TcHmiSymbol.Show'}
    rot : LREAL;
    {attribute 'TcHmiSymbol.Show'}
    roc : LREAL;
    {attribute 'TcHmiSymbol.Show'}
    ron : LREAL;
    {attribute 'TcHmiSymbol.Show'}
    doAzi : BOOL;
    {attribute 'TcHmiSymbol.Show'}
    doEle : BOOL;
    {attribute 'TcHmiSymbol.Show'}
    doRot : BOOL;
    {attribute 'TcHmiSymbol.Show'}
    doRoc : BOOL;
    {attribute 'TcHmiSymbol.Show'}
    doRon : BOOL;
    {attribute 'TcHmiSymbol.Show'}
    preferMostTravel : BOOL;
  END_VAR
                  moveRelative := THIS^.processes.moveRelative.request(
    units := units,
    azi := azi,
    ele := ele,
    rot := rot,
    roc := roc,
    ron := ron,
    doAzi := doAzi,
    doEle := doEle,
    doRot := doRot,
    doRoc := doRoc,
    doRon := doRon,
    preferMostTravel := preferMostTravel);

                
END_METHOD

{attribute 'TcRpcEnable' := '1'}
METHOD moveKnownPosition : RequestResults
  VAR_INPUT
    {attribute 'TcHmiSymbol.Show'}
    name : STRING;
  END_VAR
                  moveKnownPosition := THIS^.processes.moveKnownPosition.request( name := name );

                
END_METHOD

{attribute 'TcRpcEnable' := '1'}
METHOD enablePointingModel : RequestResults
  VAR_INPUT
    {attribute 'TcHmiSymbol.Show'}
    name : STRING;
  END_VAR
                  enablePointingModel := THIS^.processes.enablePointingModel.request( name := name );

                
END_METHOD

{attribute 'TcRpcEnable' := '1'}
METHOD disablePointingModel : RequestResults
                  disablePointingModel := THIS^.processes.disablePointingModel.request();

                
END_METHOD

{attribute 'TcRpcEnable' := '1'}
METHOD setAlphaDeltaVelocity : RequestResults
  VAR_INPUT
    {attribute 'TcHmiSymbol.Show'}
    units : AxesMoveVelocityUnits;
    {attribute 'TcHmiSymbol.Show'}
    alphaVelocity : LREAL;
    {attribute 'TcHmiSymbol.Show'}
    deltaVelocity : LREAL;
  END_VAR
                  setAlphaDeltaVelocity := THIS^.processes.setAlphaDeltaVelocity.request(
    units := units,
    alphaVelocity := alphaVelocity,
    deltaVelocity := deltaVelocity);

                
END_METHOD

METHOD _log : BOOL
  VAR_INPUT
    {attribute 'TcHmiSymbol.Show'}
    name : STRING;  (* Name of this function block instance *)
  END_VAR
  VAR_IN_OUT
    {attribute 'TcHmiSymbol.Show'}
    buffer : LogBuffer;  (* Buffer to write all logging to *)
  END_VAR
  VAR
    {attribute 'TcHmiSymbol.Show'}
    subBuffer : LogBuffer;  (* Temporary buffer to write logging by parts (sub-statemachines) to *)
  END_VAR
                  THIS^.parts.azi._log(
    name := 'azi',
    buffer := subBuffer);
THIS^.parts.ele._log(
    name := 'ele',
    buffer := subBuffer);
THIS^.parts.roc._log(
    name := 'roc',
    buffer := subBuffer);
THIS^.parts.ron._log(
    name := 'ron',
    buffer := subBuffer);
THIS^.parts.io._log(
    name := 'io',
    buffer := subBuffer);
THIS^.parts.configManager._log(
    name := 'configManager',
    buffer := subBuffer);
THIS^.parts.tpoint._log(
    name := 'tpoint',
    buffer := subBuffer);
THIS^.processes.initialize._log(
    name := 'processes.initialize',
    buffer := subBuffer);
THIS^.processes.reset._log(
    name := 'processes.reset',
    buffer := subBuffer);
THIS^.processes.lock._log(
    name := 'processes.lock',
    buffer := subBuffer);
THIS^.processes.unlock._log(
    name := 'processes.unlock',
    buffer := subBuffer);
THIS^.processes.changeOperatingState._log(
    name := 'processes.changeOperatingState',
    buffer := subBuffer);
THIS^.processes.setTarget._log(
    name := 'processes.setTarget',
    buffer := subBuffer);
THIS^.processes.point._log(
    name := 'processes.point',
    buffer := subBuffer);
THIS^.processes.pointRelative._log(
    name := 'processes.pointRelative',
    buffer := subBuffer);
THIS^.processes.stop._log(
    name := 'processes.stop',
    buffer := subBuffer);
THIS^.processes.quickStop._log(
    name := 'processes.quickStop',
    buffer := subBuffer);
THIS^.processes.powerOn._log(
    name := 'processes.powerOn',
    buffer := subBuffer);
THIS^.processes.powerOff._log(
    name := 'processes.powerOff',
    buffer := subBuffer);
THIS^.processes.doHoming._log(
    name := 'processes.doHoming',
    buffer := subBuffer);
THIS^.processes.moveAbsolute._log(
    name := 'processes.moveAbsolute',
    buffer := subBuffer);
THIS^.processes.moveRelative._log(
    name := 'processes.moveRelative',
    buffer := subBuffer);
THIS^.processes.moveKnownPosition._log(
    name := 'processes.moveKnownPosition',
    buffer := subBuffer);
THIS^.processes.enablePointingModel._log(
    name := 'processes.enablePointingModel',
    buffer := subBuffer);
THIS^.processes.disablePointingModel._log(
    name := 'processes.disablePointingModel',
    buffer := subBuffer);
THIS^.processes.setAlphaDeltaVelocity._log(
    name := 'processes.setAlphaDeltaVelocity',
    buffer := subBuffer);
LOGGER(
    name := name,
    actualStatus := THIS^.actualStatus,
    previousStatus := THIS^.previousStatus,
    buffer := buffer,
    subBuffer := subBuffer,
    pHealthStatus := ADR(THIS^.statuses.healthStatus),
    pBusyStatus := ADR(THIS^.statuses.busyStatus));

                
END_METHOD
END_FUNCTION_BLOCK

FUNCTION_BLOCK SM_AxesTarget
  VAR_INPUT
    {attribute 'TcHmiSymbol.Show'}
    {attribute 'OPC.UA.DA' := '1'}
    {attribute 'OPC.UA.DA.Access' := '1'}
    isGiven : BOOL;  (* True if the target is given, false if not *)
    {attribute 'TcHmiSymbol.Show'}
    {attribute 'OPC.UA.DA' := '1'}
    {attribute 'OPC.UA.DA.Access' := '1'}
    isValid : BOOL;  (* True if the target is valid, false if not *)
    {attribute 'TcHmiSymbol.Show'}
    {attribute 'OPC.UA.DA' := '1'}
    {attribute 'OPC.UA.DA.Access' := '1'}
    isTooLow : BOOL;  (* True if the target is too low to calculate, false if not *)
    {attribute 'TcHmiSymbol.Show'}
    {attribute 'OPC.UA.DA' := '1'}
    {attribute 'OPC.UA.DA.Access' := '1'}
    alpha : AngularPosition;  (* The alpha coordinate (Right Ascention) *)
    {attribute 'TcHmiSymbol.Show'}
    {attribute 'OPC.UA.DA' := '1'}
    {attribute 'OPC.UA.DA.Access' := '1'}
    delta : AngularPosition;  (* The delta coordinate (Declination) *)
    {attribute 'TcHmiSymbol.Show'}
    {attribute 'OPC.UA.DA' := '1'}
    {attribute 'OPC.UA.DA.Access' := '1'}
    muAlpha : LREAL;  (* Right ascention proper motion, in arcseconds/year (not multiplied by cos(delta)!) *)
    {attribute 'TcHmiSymbol.Show'}
    {attribute 'OPC.UA.DA' := '1'}
    {attribute 'OPC.UA.DA.Access' := '1'}
    muDelta : LREAL;  (* Declination proper motion, in arcseconds/year *)
    {attribute 'TcHmiSymbol.Show'}
    {attribute 'OPC.UA.DA' := '1'}
    {attribute 'OPC.UA.DA.Access' := '1'}
    parallax : LREAL;  (* Object parallax, in arcseconds *)
    {attribute 'TcHmiSymbol.Show'}
    {attribute 'OPC.UA.DA' := '1'}
    {attribute 'OPC.UA.DA.Access' := '1'}
    radialVelocity : LREAL;  (* Object radial velocity, in km/s *)
    {attribute 'TcHmiSymbol.Show'}
    {attribute 'OPC.UA.DA' := '1'}
    {attribute 'OPC.UA.DA.Access' := '1'}
    epoch : LREAL;  (* Epoch, e.g. 2000.0 *)
    {attribute 'TcHmiSymbol.Show'}
    {attribute 'OPC.UA.DA' := '1'}
    {attribute 'OPC.UA.DA.Access' := '1'}
    alphaVelocity : AngularVelocity;  (* Additional target velocity (e.g. for solar system objects) in alpha direction *)
    {attribute 'TcHmiSymbol.Show'}
    {attribute 'OPC.UA.DA' := '1'}
    {attribute 'OPC.UA.DA.Access' := '1'}
    deltaVelocity : AngularVelocity;  (* Additional target velocity (e.g. for solar system objects) in delta direction *)
    {attribute 'TcHmiSymbol.Show'}
    {attribute 'OPC.UA.DA' := '1'}
    {attribute 'OPC.UA.DA.Access' := '1'}
    alphaTravelled : AngularPosition;  (* Alpha traveled so far due to the alphaVelocity *)
    {attribute 'TcHmiSymbol.Show'}
    {attribute 'OPC.UA.DA' := '1'}
    {attribute 'OPC.UA.DA.Access' := '1'}
    deltaTravelled : AngularPosition;  (* Delta traveled so far due to the deltaVelocity *)
    {attribute 'TcHmiSymbol.Show'}
    {attribute 'OPC.UA.DA' := '1'}
    {attribute 'OPC.UA.DA.Access' := '1'}
    alphaOffsetted : AngularPosition;  (* Alpha offsetted so far due to the alphaOffset *)
    {attribute 'TcHmiSymbol.Show'}
    {attribute 'OPC.UA.DA' := '1'}
    {attribute 'OPC.UA.DA.Access' := '1'}
    deltaOffsetted : AngularPosition;  (* Delta offsetted so far due to the deltaOffset *)
    {attribute 'TcHmiSymbol.Show'}
    {attribute 'OPC.UA.DA' := '1'}
    {attribute 'OPC.UA.DA.Access' := '1'}
    alphaStart : AngularPosition;  (* Original alpha without traveling (=alpha - alphaTraveled - alphaOffsetted) *)
    {attribute 'TcHmiSymbol.Show'}
    {attribute 'OPC.UA.DA' := '1'}
    {attribute 'OPC.UA.DA.Access' := '1'}
    deltaStart : AngularPosition;  (* Original delta without traveling (=delta - deltaTraveled - deltaOffsetted) *)
    {attribute 'TcHmiSymbol.Show'}
    {attribute 'OPC.UA.DA' := '1'}
    {attribute 'OPC.UA.DA.Access' := '1'}
    aziPos : AngularPosition;  (* The azimuth target position, as calculated by SLALIBl *)
    {attribute 'TcHmiSymbol.Show'}
    {attribute 'OPC.UA.DA' := '1'}
    {attribute 'OPC.UA.DA.Access' := '1'}
    aziVelo : AngularVelocity;  (* The azimuth target velocity, as calculated by SLALIB *)
    {attribute 'TcHmiSymbol.Show'}
    {attribute 'OPC.UA.DA' := '1'}
    {attribute 'OPC.UA.DA.Access' := '1'}
    aziAcc : AngularAcceleration;  (* The azimuth target acceleration, as calculated by SLALIB *)
    {attribute 'TcHmiSymbol.Show'}
    {attribute 'OPC.UA.DA' := '1'}
    {attribute 'OPC.UA.DA.Access' := '1'}
    elePos : AngularPosition;  (* The elevation target position, as calculated by SLALIB *)
    {attribute 'TcHmiSymbol.Show'}
    {attribute 'OPC.UA.DA' := '1'}
    {attribute 'OPC.UA.DA.Access' := '1'}
    eleVelo : AngularVelocity;  (* The elevation target velocity, as calculated by SLALIB *)
    {attribute 'TcHmiSymbol.Show'}
    {attribute 'OPC.UA.DA' := '1'}
    {attribute 'OPC.UA.DA.Access' := '1'}
    eleAcc : AngularAcceleration;  (* The elevation target acceleration, as calculated by SLALIB *)
    {attribute 'TcHmiSymbol.Show'}
    {attribute 'OPC.UA.DA' := '1'}
    {attribute 'OPC.UA.DA.Access' := '1'}
    paPos : AngularPosition;  (* The position angle target position, as calculated by SLALIB *)
    {attribute 'TcHmiSymbol.Show'}
    {attribute 'OPC.UA.DA' := '1'}
    {attribute 'OPC.UA.DA.Access' := '1'}
    paVelo : AngularVelocity;  (* The position angle target velocity, as calculated by SLALIB *)
    {attribute 'TcHmiSymbol.Show'}
    {attribute 'OPC.UA.DA' := '1'}
    {attribute 'OPC.UA.DA.Access' := '1'}
    paAcc : AngularAcceleration;  (* The position angle target acceleration, as calculated by SLALIB *)
    {attribute 'TcHmiSymbol.Show'}
    {attribute 'OPC.UA.DA' := '1'}
    {attribute 'OPC.UA.DA.Access' := '1'}
    aziPointingModelOffset : AngularPosition;  (* The azimuth pointing model offset calculated by the TPoint model *)
    {attribute 'TcHmiSymbol.Show'}
    {attribute 'OPC.UA.DA' := '1'}
    {attribute 'OPC.UA.DA.Access' := '1'}
    elePointingModelOffset : AngularPosition;  (* The elevation pointing model offset calculated by the TPoint model *)
    {attribute 'TcHmiSymbol.Show'}
    {attribute 'OPC.UA.DA' := '1'}
    {attribute 'OPC.UA.DA.Access' := '1'}
    correctedAzi : AngularPosition;  (* The azimuth target position, as calculated by SLALIB, corrected by the TPoint model *)
    {attribute 'TcHmiSymbol.Show'}
    {attribute 'OPC.UA.DA' := '1'}
    {attribute 'OPC.UA.DA.Access' := '1'}
    correctedEle : AngularPosition;  (* The elevation target position, as calculated by SLALIB, corrected by the TPoint model *)
  END_VAR
  VAR_OUTPUT
    {attribute 'OPC.UA.DA' := '1'}
    {attribute 'OPC.UA.DA.Access' := '1'}
    {attribute 'TcHmiSymbol.Show'}
    actualStatus : STRING;  (* Current status description *)
    {attribute 'TcHmiSymbol.Show'}
    previousStatus : STRING;  (* Previous status description *)
    {attribute 'TcHmiSymbol.Show'}
    statuses : AxesTargetStatuses;  (* Statuses of the state machine *)
  END_VAR

            statuses.healthStatus( isGood := isValid OR (NOT(isGiven)) );

          

METHOD _log : BOOL
  VAR_INPUT
    {attribute 'TcHmiSymbol.Show'}
    name : STRING;  (* Name of this function block instance *)
  END_VAR
  VAR_IN_OUT
    {attribute 'TcHmiSymbol.Show'}
    buffer : LogBuffer;  (* Buffer to write all logging to *)
  END_VAR
  VAR
    {attribute 'TcHmiSymbol.Show'}
    subBuffer : LogBuffer;  (* Temporary buffer to write logging by parts (sub-statemachines) to *)
  END_VAR
                  LOGGER(
    name := name,
    actualStatus := THIS^.actualStatus,
    previousStatus := THIS^.previousStatus,
    buffer := buffer,
    subBuffer := subBuffer,
    pHealthStatus := ADR(THIS^.statuses.healthStatus));

                
END_METHOD
END_FUNCTION_BLOCK

FUNCTION_BLOCK SM_AxesFeedback
  VAR_INPUT
    {attribute 'TcHmiSymbol.Show'}
    {attribute 'OPC.UA.DA' := '1'}
    {attribute 'OPC.UA.DA.Access' := '1'}
    isValid : BOOL;  (* True if the feedback is valid, false if not *)
    {attribute 'TcHmiSymbol.Show'}
    {attribute 'OPC.UA.DA' := '1'}
    {attribute 'OPC.UA.DA.Access' := '1'}
    isTooLow : BOOL;  (* True if the feedback is too low to calculate, false if not *)
    {attribute 'TcHmiSymbol.Show'}
    {attribute 'OPC.UA.DA' := '1'}
    {attribute 'OPC.UA.DA.Access' := '1'}
    alpha : AngularPosition;  (* The alpha coordinate (Right Ascention) *)
    {attribute 'TcHmiSymbol.Show'}
    {attribute 'OPC.UA.DA' := '1'}
    {attribute 'OPC.UA.DA.Access' := '1'}
    delta : AngularPosition;  (* The delta coordinate (Declination) *)
    {attribute 'TcHmiSymbol.Show'}
    {attribute 'OPC.UA.DA' := '1'}
    {attribute 'OPC.UA.DA.Access' := '1'}
    aziPos : AngularPosition;  (* The measured AZI position, corrected by TPoint, and normalized to [0..2*PI] *)
    {attribute 'TcHmiSymbol.Show'}
    {attribute 'OPC.UA.DA' := '1'}
    {attribute 'OPC.UA.DA.Access' := '1'}
    elePos : AngularPosition;  (* The measured ELE position, corrected by TPoint, normalized to [-PI..PI] *)
    {attribute 'TcHmiSymbol.Show'}
    {attribute 'OPC.UA.DA' := '1'}
    {attribute 'OPC.UA.DA.Access' := '1'}
    rocPos : AngularPosition;  (* The measured ROC position, normalized to [-PI..PI] *)
    {attribute 'TcHmiSymbol.Show'}
    {attribute 'OPC.UA.DA' := '1'}
    {attribute 'OPC.UA.DA.Access' := '1'}
    ronPos : AngularPosition;  (* The measured RON position, normalized to [-PI..PI] *)
    {attribute 'TcHmiSymbol.Show'}
    {attribute 'OPC.UA.DA' := '1'}
    {attribute 'OPC.UA.DA.Access' := '1'}
    rotPos : AngularPosition;  (* The measured position of the currently active rotator (ROC or RON), normalized to [-PI..PI] *)
    {attribute 'TcHmiSymbol.Show'}
    {attribute 'OPC.UA.DA' := '1'}
    {attribute 'OPC.UA.DA.Access' := '1'}
    rotOffset : AngularPosition;  (* The active rotator offset, to North *)
    {attribute 'TcHmiSymbol.Show'}
    {attribute 'OPC.UA.DA' := '1'}
    {attribute 'OPC.UA.DA.Access' := '1'}
    rocOffset : AngularPosition;  (* The cassegrain rotator offset, to North *)
    {attribute 'TcHmiSymbol.Show'}
    {attribute 'OPC.UA.DA' := '1'}
    {attribute 'OPC.UA.DA.Access' := '1'}
    ronOffset : AngularPosition;  (* The nasmyth rotator offset, to North *)
  END_VAR
  VAR_OUTPUT
    {attribute 'OPC.UA.DA' := '1'}
    {attribute 'OPC.UA.DA.Access' := '1'}
    {attribute 'TcHmiSymbol.Show'}
    actualStatus : STRING;  (* Current status description *)
    {attribute 'TcHmiSymbol.Show'}
    previousStatus : STRING;  (* Previous status description *)
    {attribute 'TcHmiSymbol.Show'}
    statuses : AxesFeedbackStatuses;  (* Statuses of the state machine *)
  END_VAR

            statuses.healthStatus( isGood := isValid );

          

METHOD _log : BOOL
  VAR_INPUT
    {attribute 'TcHmiSymbol.Show'}
    name : STRING;  (* Name of this function block instance *)
  END_VAR
  VAR_IN_OUT
    {attribute 'TcHmiSymbol.Show'}
    buffer : LogBuffer;  (* Buffer to write all logging to *)
  END_VAR
  VAR
    {attribute 'TcHmiSymbol.Show'}
    subBuffer : LogBuffer;  (* Temporary buffer to write logging by parts (sub-statemachines) to *)
  END_VAR
                  LOGGER(
    name := name,
    actualStatus := THIS^.actualStatus,
    previousStatus := THIS^.previousStatus,
    buffer := buffer,
    subBuffer := subBuffer,
    pHealthStatus := ADR(THIS^.statuses.healthStatus));

                
END_METHOD
END_FUNCTION_BLOCK

FUNCTION_BLOCK SM_AxesAzimuthAxis
  VAR_INPUT
    {attribute 'TcHmiSymbol.Show'}
    {attribute 'OPC.UA.DA' := '1'}
    {attribute 'OPC.UA.DA.Access' := '1'}
    id : AxesIds;  (* Id of this axis *)
    {attribute 'TcHmiSymbol.Show'}
    {attribute 'OPC.UA.DA' := '0'}
    {attribute 'TcHmiSymbol.Hide'}
    isEnabled : BOOL;  (* Is control enabled? *)
    {attribute 'TcHmiSymbol.Show'}
    {attribute 'OPC.UA.DA' := '0'}
    {attribute 'TcHmiSymbol.Hide'}
    REDUCTION_AZI_TO_TEL : LREAL := 1440.0;  (* The mechanical reduction between absolute encoder and telescope *)
    {attribute 'TcHmiSymbol.Show'}
    {attribute 'OPC.UA.DA' := '0'}
    {attribute 'TcHmiSymbol.Hide'}
    REDUCTION_ABL_TO_TEL : LREAL := 180.0;  (* The mechanical reduction between absolute encoder and telescope *)
    {attribute 'TcHmiSymbol.Show'}
    {attribute 'OPC.UA.DA' := '0'}
    {attribute 'TcHmiSymbol.Hide'}
    REDUCTION_ABS_ENC_TO_TEL : LREAL := 18.0;  (* The mechanical reduction between absolute encoder and telescope *)
  END_VAR
  VAR_OUTPUT
    {attribute 'OPC.UA.DA' := '1'}
    {attribute 'OPC.UA.DA.Access' := '1'}
    {attribute 'TcHmiSymbol.Show'}
    actualStatus : STRING;  (* Current status description *)
    {attribute 'TcHmiSymbol.Show'}
    previousStatus : STRING;  (* Previous status description *)
    {attribute 'TcHmiSymbol.Show'}
    {attribute 'OPC.UA.DA' := '1'}
    {attribute 'OPC.UA.DA.Access' := '1'}
    slipError : BOOL;  (* TRUE if the motor appears to be slipping w.r.t. the external encoder *)
    {attribute 'TcHmiSymbol.Show'}
    {attribute 'OPC.UA.DA' := '1'}
    {attribute 'OPC.UA.DA.Access' := '1'}
    positiveLimitSwitchError : BOOL;  (* TRUE if the positive limit switch has detected the axis *)
    {attribute 'TcHmiSymbol.Show'}
    {attribute 'OPC.UA.DA' := '1'}
    {attribute 'OPC.UA.DA.Access' := '1'}
    negativeLimitSwitchError : BOOL;  (* TRUE if the negative limit switch has detected the axis *)
    {attribute 'TcHmiSymbol.Show'}
    {attribute 'OPC.UA.DA' := '1'}
    {attribute 'OPC.UA.DA.Access' := '1'}
    setPosLimitReached : BOOL;  (* TRUE if the setpoint position has reached its limit *)
    {attribute 'TcHmiSymbol.Show'}
    {attribute 'OPC.UA.DA' := '1'}
    {attribute 'OPC.UA.DA.Access' := '1'}
    deviation1SecAverage : AngularPosition;  (* The deviation between target position and actual position, as a 1 second moving average *)
    {attribute 'TcHmiSymbol.Show'}
    {attribute 'OPC.UA.DA' := '1'}
    {attribute 'OPC.UA.DA.Access' := '1'}
    deviation1SecRMS : AngularPosition;  (* The deviation between target position and actual position, as a 1 second moving RMS error *)
    {attribute 'TcHmiSymbol.Show'}
    {attribute 'OPC.UA.DA' := '1'}
    {attribute 'OPC.UA.DA.Access' := '1'}
    targetPos : AngularPosition;  (* The target position *)
    {attribute 'TcHmiSymbol.Show'}
    {attribute 'OPC.UA.DA' := '1'}
    {attribute 'OPC.UA.DA.Access' := '1'}
    targetOffset : AngularPosition;  (* Cumulative offset of targetPos. Equals targetPos - targetStart *)
    {attribute 'TcHmiSymbol.Show'}
    {attribute 'OPC.UA.DA' := '1'}
    {attribute 'OPC.UA.DA.Access' := '1'}
    targetStart : AngularPosition;  (* Last absolute movement end position of the axis *)
    {attribute 'TcHmiSymbol.Show'}
    {attribute 'OPC.UA.DA' := '1'}
    {attribute 'OPC.UA.DA.Access' := '1'}
    setPos : AngularPosition;  (* The setpoint position (same as parts.physicalAxis!) *)
    {attribute 'TcHmiSymbol.Show'}
    {attribute 'OPC.UA.DA' := '1'}
    {attribute 'OPC.UA.DA.Access' := '1'}
    setVelo : AngularVelocity;  (* The setpoint velocity (same as parts.physicalAxis!) *)
    {attribute 'TcHmiSymbol.Show'}
    {attribute 'OPC.UA.DA' := '1'}
    {attribute 'OPC.UA.DA.Access' := '1'}
    setAcc : AngularAcceleration;  (* The setpoint acceleration (same as parts.physicalAxis!) *)
    {attribute 'TcHmiSymbol.Show'}
    {attribute 'OPC.UA.DA' := '1'}
    {attribute 'OPC.UA.DA.Access' := '1'}
    actPos : AngularPosition;  (* The actual position (same as parts.physicalAxis!) *)
    {attribute 'TcHmiSymbol.Show'}
    {attribute 'OPC.UA.DA' := '1'}
    {attribute 'OPC.UA.DA.Access' := '1'}
    actVelo : AngularVelocity;  (* The actual velocity (same as parts.physicalAxis!) *)
    {attribute 'TcHmiSymbol.Show'}
    {attribute 'OPC.UA.DA' := '1'}
    {attribute 'OPC.UA.DA.Access' := '1'}
    actAcc : AngularAcceleration;  (* The actual acceleration (same as parts.physicalAxis!) *)
    {attribute 'TcHmiSymbol.Show'}
    {attribute 'OPC.UA.DA' := '1'}
    {attribute 'OPC.UA.DA.Access' := '1'}
    actTorqueAzi : Torque;  (* The actual torque on the telescope axis by the AZI motor *)
    {attribute 'TcHmiSymbol.Show'}
    {attribute 'OPC.UA.DA' := '1'}
    {attribute 'OPC.UA.DA.Access' := '1'}
    actTorqueAbl : Torque;  (* The actual torque on the telescope axis by the ABL motor *)
    {attribute 'TcHmiSymbol.Show'}
    {attribute 'OPC.UA.DA' := '1'}
    {attribute 'OPC.UA.DA.Access' := '1'}
    lida1Position : AngularPosition;  (* Position of the telescope according to LIDA encoder no. 1 *)
    {attribute 'TcHmiSymbol.Show'}
    {attribute 'OPC.UA.DA' := '1'}
    {attribute 'OPC.UA.DA.Access' := '1'}
    lida2Position : AngularPosition;  (* Position of the telescope according to LIDA encoder no. 2 *)
    {attribute 'TcHmiSymbol.Show'}
    {attribute 'OPC.UA.DA' := '1'}
    {attribute 'OPC.UA.DA.Access' := '1'}
    lida3Position : AngularPosition;  (* Position of the telescope according to LIDA encoder no. 3 *)
    {attribute 'TcHmiSymbol.Show'}
    {attribute 'OPC.UA.DA' := '1'}
    {attribute 'OPC.UA.DA.Access' := '1'}
    lida4Position : AngularPosition;  (* Position of the telescope according to LIDA encoder no. 4 *)
    {attribute 'TcHmiSymbol.Show'}
    {attribute 'OPC.UA.DA' := '1'}
    {attribute 'OPC.UA.DA.Access' := '1'}
    lidaAveragePosition : AngularPosition;  (* Position of the telescope according to the average of the LIDA encoders *)
    {attribute 'TcHmiSymbol.Show'}
    {attribute 'OPC.UA.DA' := '1'}
    {attribute 'OPC.UA.DA.Access' := '1'}
    absoluteEncoderPosition : AngularPosition;  (* The position of the axis, based on the absolute encoder *)
    {attribute 'TcHmiSymbol.Show'}
    statuses : AxesAzimuthAxisStatuses;  (* Statuses of the state machine *)
    {attribute 'TcHmiSymbol.Show'}
    parts : AxesAzimuthAxisParts;  (* Parts of the state machine *)
    {attribute 'TcHmiSymbol.Show'}
    processes : AxesAzimuthAxisProcesses;  (* Processes of the state machine *)
  END_VAR
  VAR_IN_OUT
    {attribute 'TcHmiSymbol.Show'}
    {attribute 'OPC.UA.DA' := '0'}
    {attribute 'TcHmiSymbol.Hide'}
    config : AxesAzimuthConfig;  (* Reference to the azimuth config *)
    {attribute 'TcHmiSymbol.Show'}
    {attribute 'OPC.UA.DA' := '0'}
    {attribute 'TcHmiSymbol.Hide'}
    aziDriveChannel : AX52XXDriveChannel;  (* Reference to the AZI drive channel *)
    {attribute 'TcHmiSymbol.Show'}
    {attribute 'OPC.UA.DA' := '0'}
    {attribute 'TcHmiSymbol.Hide'}
    ablDriveChannel : AX52XXDriveChannel;  (* Reference to the ABL drive channel *)
    {attribute 'TcHmiSymbol.Show'}
    {attribute 'OPC.UA.DA' := '0'}
    {attribute 'TcHmiSymbol.Hide'}
    aziMainDriveChannel : AX52XXDriveChannel;  (* Reference to the main drive channel (channel A) of the drive *)
    {attribute 'TcHmiSymbol.Show'}
    {attribute 'OPC.UA.DA' := '0'}
    {attribute 'TcHmiSymbol.Hide'}
    ablMainDriveChannel : AX52XXDriveChannel;  (* Reference to the main drive channel (channel A) of the drive *)
  END_VAR

            parts.virtualAxis( isEnabled := isEnabled );
parts.physicalAxis( isEnabled := isEnabled );
parts.ablAxis( isEnabled := isEnabled );
parts.lida1( isEnabled := isEnabled );
parts.lida2( isEnabled := isEnabled );
parts.lida3( isEnabled := isEnabled );
parts.lida4( isEnabled := isEnabled );
parts.absoluteEncoder();
statuses.busyStatus( isBusy := aziDriveChannel.statuses.busyStatus.busy OR (ablDriveChannel.statuses.busyStatus.busy OR (parts.virtualAxis.statuses.busyStatus.busy OR (parts.physicalAxis.statuses.busyStatus.busy OR (parts.ablAxis.statuses.busyStatus.busy OR (parts.lida1.statuses.busyStatus.busy OR (parts.lida2.statuses.busyStatus.busy OR (parts.lida3.statuses.busyStatus.busy OR (parts.lida4.statuses.busyStatus.busy OR (processes.moveAbsolute.statuses.busyStatus.busy OR (processes.moveRelative.statuses.busyStatus.busy OR (processes.moveVelocity.statuses.busyStatus.busy OR (processes.reset.statuses.busyStatus.busy OR (processes.moveOutOfLimitSwitch.statuses.busyStatus.busy OR (processes.powerOn.statuses.busyStatus.busy OR (processes.powerOff.statuses.busyStatus.busy OR (processes.doHoming.statuses.busyStatus.busy OR (processes.stop.statuses.busyStatus.busy OR (processes.quickStop.statuses.busyStatus.busy OR (processes.unlockBrake.statuses.busyStatus.busy OR processes.setPosition.statuses.busyStatus.busy))))))))))))))))))) );
statuses.healthStatus(
    isGood := (aziDriveChannel.statuses.healthStatus.isGood AND (ablDriveChannel.statuses.healthStatus.isGood AND (parts.virtualAxis.statuses.healthStatus.isGood AND (parts.physicalAxis.statuses.healthStatus.isGood AND (parts.ablAxis.statuses.healthStatus.isGood AND (parts.lida1.statuses.healthStatus.isGood AND (parts.lida2.statuses.healthStatus.isGood AND (parts.lida3.statuses.healthStatus.isGood AND (parts.lida4.statuses.healthStatus.isGood AND (parts.absoluteEncoder.statuses.healthStatus.isGood AND (processes.moveAbsolute.statuses.healthStatus.isGood AND (processes.moveRelative.statuses.healthStatus.isGood AND (processes.moveVelocity.statuses.healthStatus.isGood AND (processes.reset.statuses.healthStatus.isGood AND (processes.moveOutOfLimitSwitch.statuses.healthStatus.isGood AND (processes.powerOn.statuses.healthStatus.isGood AND (processes.powerOff.statuses.healthStatus.isGood AND (processes.doHoming.statuses.healthStatus.isGood AND (processes.stop.statuses.healthStatus.isGood AND (processes.quickStop.statuses.healthStatus.isGood AND (processes.unlockBrake.statuses.healthStatus.isGood AND processes.setPosition.statuses.healthStatus.isGood))))))))))))))))))))) AND ((NOT(slipError)) AND ((NOT(positiveLimitSwitchError)) AND (NOT(negativeLimitSwitchError)))),
    hasWarning := aziDriveChannel.statuses.healthStatus.hasWarning OR (ablDriveChannel.statuses.healthStatus.hasWarning OR (parts.virtualAxis.statuses.healthStatus.hasWarning OR (parts.physicalAxis.statuses.healthStatus.hasWarning OR (parts.ablAxis.statuses.healthStatus.hasWarning OR (parts.lida1.statuses.healthStatus.hasWarning OR (parts.lida2.statuses.healthStatus.hasWarning OR (parts.lida3.statuses.healthStatus.hasWarning OR (parts.lida4.statuses.healthStatus.hasWarning OR (parts.absoluteEncoder.statuses.healthStatus.hasWarning OR (processes.moveAbsolute.statuses.healthStatus.hasWarning OR (processes.moveRelative.statuses.healthStatus.hasWarning OR (processes.moveVelocity.statuses.healthStatus.hasWarning OR (processes.reset.statuses.healthStatus.hasWarning OR (processes.moveOutOfLimitSwitch.statuses.healthStatus.hasWarning OR (processes.powerOn.statuses.healthStatus.hasWarning OR (processes.powerOff.statuses.healthStatus.hasWarning OR (processes.doHoming.statuses.healthStatus.hasWarning OR (processes.stop.statuses.healthStatus.hasWarning OR (processes.quickStop.statuses.healthStatus.hasWarning OR (processes.unlockBrake.statuses.healthStatus.hasWarning OR processes.setPosition.statuses.healthStatus.hasWarning)))))))))))))))))))));
statuses.poweredStatus( isEnabled := parts.virtualAxis.statuses.poweredStatus.enabled AND (parts.physicalAxis.statuses.poweredStatus.enabled AND parts.ablAxis.statuses.poweredStatus.enabled) );
processes.moveAbsolute( isEnabled := isEnabled );
processes.moveRelative( isEnabled := isEnabled );
processes.moveVelocity( isEnabled := isEnabled );
processes.reset( isEnabled := isEnabled );
processes.moveOutOfLimitSwitch( isEnabled := isEnabled );
processes.powerOn( isEnabled := isEnabled );
processes.powerOff( isEnabled := isEnabled );
processes.doHoming( isEnabled := isEnabled );
processes.stop( isEnabled := isEnabled );
processes.quickStop( isEnabled := isEnabled );
processes.unlockBrake( isEnabled := isEnabled );
processes.setPosition( isEnabled := isEnabled );

          

{attribute 'TcRpcEnable' := '1'}
METHOD moveAbsolute : RequestResults
  VAR_INPUT
    {attribute 'TcHmiSymbol.Show'}
    units : AxesMoveUnits;
    {attribute 'TcHmiSymbol.Show'}
    value : LREAL;
    {attribute 'TcHmiSymbol.Show'}
    offset : LREAL;
  END_VAR
                  moveAbsolute := THIS^.processes.moveAbsolute.request(
    units := units,
    value := value,
    offset := offset);

                
END_METHOD

{attribute 'TcRpcEnable' := '1'}
METHOD moveRelative : RequestResults
  VAR_INPUT
    {attribute 'TcHmiSymbol.Show'}
    units : AxesMoveUnits;
    {attribute 'TcHmiSymbol.Show'}
    value : LREAL;
  END_VAR
                  moveRelative := THIS^.processes.moveRelative.request(
    units := units,
    value := value);

                
END_METHOD

{attribute 'TcRpcEnable' := '1'}
METHOD moveVelocity : RequestResults
  VAR_INPUT
    {attribute 'TcHmiSymbol.Show'}
    units : AxesMoveVelocityUnits;
    {attribute 'TcHmiSymbol.Show'}
    value : LREAL;
  END_VAR
                  moveVelocity := THIS^.processes.moveVelocity.request(
    units := units,
    value := value);

                
END_METHOD

{attribute 'TcRpcEnable' := '1'}
METHOD reset : RequestResults
                  reset := THIS^.processes.reset.request();

                
END_METHOD

{attribute 'TcRpcEnable' := '1'}
METHOD moveOutOfLimitSwitch : RequestResults
  VAR_INPUT
    {attribute 'TcHmiSymbol.Show'}
    switch : LimitSwitches;
  END_VAR
                  moveOutOfLimitSwitch := THIS^.processes.moveOutOfLimitSwitch.request( switch := switch );

                
END_METHOD

{attribute 'TcRpcEnable' := '1'}
METHOD powerOn : RequestResults
                  powerOn := THIS^.processes.powerOn.request();

                
END_METHOD

{attribute 'TcRpcEnable' := '1'}
METHOD powerOff : RequestResults
                  powerOff := THIS^.processes.powerOff.request();

                
END_METHOD

{attribute 'TcRpcEnable' := '1'}
METHOD doHoming : RequestResults
                  doHoming := THIS^.processes.doHoming.request();

                
END_METHOD

{attribute 'TcRpcEnable' := '1'}
METHOD stop : RequestResults
                  stop := THIS^.processes.stop.request();

                
END_METHOD

{attribute 'TcRpcEnable' := '1'}
METHOD quickStop : RequestResults
                  quickStop := THIS^.processes.quickStop.request();

                
END_METHOD

{attribute 'TcRpcEnable' := '1'}
METHOD unlockBrake : RequestResults
  VAR_INPUT
    {attribute 'TcHmiSymbol.Show'}
    seconds : LREAL;
  END_VAR
                  unlockBrake := THIS^.processes.unlockBrake.request( seconds := seconds );

                
END_METHOD

{attribute 'TcRpcEnable' := '1'}
METHOD setPosition : RequestResults
  VAR_INPUT
    {attribute 'TcHmiSymbol.Show'}
    value : LREAL;
  END_VAR
                  setPosition := THIS^.processes.setPosition.request( value := value );

                
END_METHOD

METHOD _log : BOOL
  VAR_INPUT
    {attribute 'TcHmiSymbol.Show'}
    name : STRING;  (* Name of this function block instance *)
  END_VAR
  VAR_IN_OUT
    {attribute 'TcHmiSymbol.Show'}
    buffer : LogBuffer;  (* Buffer to write all logging to *)
  END_VAR
  VAR
    {attribute 'TcHmiSymbol.Show'}
    subBuffer : LogBuffer;  (* Temporary buffer to write logging by parts (sub-statemachines) to *)
  END_VAR
                  THIS^.parts.virtualAxis._log(
    name := 'virtualAxis',
    buffer := subBuffer);
THIS^.parts.physicalAxis._log(
    name := 'physicalAxis',
    buffer := subBuffer);
THIS^.parts.ablAxis._log(
    name := 'ablAxis',
    buffer := subBuffer);
THIS^.parts.lida1._log(
    name := 'lida1',
    buffer := subBuffer);
THIS^.parts.lida2._log(
    name := 'lida2',
    buffer := subBuffer);
THIS^.parts.lida3._log(
    name := 'lida3',
    buffer := subBuffer);
THIS^.parts.lida4._log(
    name := 'lida4',
    buffer := subBuffer);
THIS^.parts.absoluteEncoder._log(
    name := 'absoluteEncoder',
    buffer := subBuffer);
THIS^.processes.moveAbsolute._log(
    name := 'processes.moveAbsolute',
    buffer := subBuffer);
THIS^.processes.moveRelative._log(
    name := 'processes.moveRelative',
    buffer := subBuffer);
THIS^.processes.moveVelocity._log(
    name := 'processes.moveVelocity',
    buffer := subBuffer);
THIS^.processes.reset._log(
    name := 'processes.reset',
    buffer := subBuffer);
THIS^.processes.moveOutOfLimitSwitch._log(
    name := 'processes.moveOutOfLimitSwitch',
    buffer := subBuffer);
THIS^.processes.powerOn._log(
    name := 'processes.powerOn',
    buffer := subBuffer);
THIS^.processes.powerOff._log(
    name := 'processes.powerOff',
    buffer := subBuffer);
THIS^.processes.doHoming._log(
    name := 'processes.doHoming',
    buffer := subBuffer);
THIS^.processes.stop._log(
    name := 'processes.stop',
    buffer := subBuffer);
THIS^.processes.quickStop._log(
    name := 'processes.quickStop',
    buffer := subBuffer);
THIS^.processes.unlockBrake._log(
    name := 'processes.unlockBrake',
    buffer := subBuffer);
THIS^.processes.setPosition._log(
    name := 'processes.setPosition',
    buffer := subBuffer);
LOGGER(
    name := name,
    actualStatus := THIS^.actualStatus,
    previousStatus := THIS^.previousStatus,
    buffer := buffer,
    subBuffer := subBuffer,
    pHealthStatus := ADR(THIS^.statuses.healthStatus),
    pBusyStatus := ADR(THIS^.statuses.busyStatus));

                
END_METHOD
END_FUNCTION_BLOCK

FUNCTION_BLOCK SM_AxesElevationAxis
  VAR_INPUT
    {attribute 'TcHmiSymbol.Show'}
    {attribute 'OPC.UA.DA' := '1'}
    {attribute 'OPC.UA.DA.Access' := '1'}
    id : AxesIds;  (* Id of this axis *)
    {attribute 'TcHmiSymbol.Show'}
    {attribute 'OPC.UA.DA' := '0'}
    {attribute 'TcHmiSymbol.Hide'}
    isEnabled : BOOL;  (* Is control enabled? *)
    {attribute 'TcHmiSymbol.Show'}
    {attribute 'OPC.UA.DA' := '0'}
    {attribute 'TcHmiSymbol.Hide'}
    REDUCTION_MOT_TO_TEL : LREAL := 1440.0;  (* The mechanical reduction between absolute encoder and telescope *)
    {attribute 'TcHmiSymbol.Show'}
    {attribute 'OPC.UA.DA' := '0'}
    {attribute 'TcHmiSymbol.Hide'}
    REDUCTION_ABS_ENC_TO_TEL : LREAL := 18.0;  (* The mechanical reduction between absolute encoder and telescope *)
  END_VAR
  VAR_OUTPUT
    {attribute 'OPC.UA.DA' := '1'}
    {attribute 'OPC.UA.DA.Access' := '1'}
    {attribute 'TcHmiSymbol.Show'}
    actualStatus : STRING;  (* Current status description *)
    {attribute 'TcHmiSymbol.Show'}
    previousStatus : STRING;  (* Previous status description *)
    {attribute 'TcHmiSymbol.Show'}
    {attribute 'OPC.UA.DA' := '1'}
    {attribute 'OPC.UA.DA.Access' := '1'}
    slipError : BOOL;  (* TRUE if the motor appears to be slipping w.r.t. the external encoder *)
    {attribute 'TcHmiSymbol.Show'}
    {attribute 'OPC.UA.DA' := '1'}
    {attribute 'OPC.UA.DA.Access' := '1'}
    positiveLimitSwitchError : BOOL;  (* TRUE if the positive limit switch has detected the axis *)
    {attribute 'TcHmiSymbol.Show'}
    {attribute 'OPC.UA.DA' := '1'}
    {attribute 'OPC.UA.DA.Access' := '1'}
    negativeLimitSwitchError : BOOL;  (* TRUE if the negative limit switch has detected the axis *)
    {attribute 'TcHmiSymbol.Show'}
    {attribute 'OPC.UA.DA' := '1'}
    {attribute 'OPC.UA.DA.Access' := '1'}
    setPosLimitReached : BOOL;  (* TRUE if the setpoint position has reached its limit *)
    {attribute 'TcHmiSymbol.Show'}
    {attribute 'OPC.UA.DA' := '1'}
    {attribute 'OPC.UA.DA.Access' := '1'}
    deviation1SecAverage : AngularPosition;  (* The deviation between target position and actual position, as a 1 second moving average *)
    {attribute 'TcHmiSymbol.Show'}
    {attribute 'OPC.UA.DA' := '1'}
    {attribute 'OPC.UA.DA.Access' := '1'}
    deviation1SecRMS : AngularPosition;  (* The deviation between target position and actual position, as a 1 second moving RMS error *)
    {attribute 'TcHmiSymbol.Show'}
    {attribute 'OPC.UA.DA' := '1'}
    {attribute 'OPC.UA.DA.Access' := '1'}
    targetPos : AngularPosition;  (* The target position *)
    {attribute 'TcHmiSymbol.Show'}
    {attribute 'OPC.UA.DA' := '1'}
    {attribute 'OPC.UA.DA.Access' := '1'}
    targetOffset : AngularPosition;  (* Cumulative offset of targetPos. Equals targetPos - targetStart *)
    {attribute 'TcHmiSymbol.Show'}
    {attribute 'OPC.UA.DA' := '1'}
    {attribute 'OPC.UA.DA.Access' := '1'}
    targetStart : AngularPosition;  (* Last absolute movement end position of the axis *)
    {attribute 'TcHmiSymbol.Show'}
    {attribute 'OPC.UA.DA' := '1'}
    {attribute 'OPC.UA.DA.Access' := '1'}
    setPos : AngularPosition;  (* The setpoint position (same as parts.physicalAxis!) *)
    {attribute 'TcHmiSymbol.Show'}
    {attribute 'OPC.UA.DA' := '1'}
    {attribute 'OPC.UA.DA.Access' := '1'}
    setVelo : AngularVelocity;  (* The setpoint velocity (same as parts.physicalAxis!) *)
    {attribute 'TcHmiSymbol.Show'}
    {attribute 'OPC.UA.DA' := '1'}
    {attribute 'OPC.UA.DA.Access' := '1'}
    setAcc : AngularAcceleration;  (* The setpoint acceleration (same as parts.physicalAxis!) *)
    {attribute 'TcHmiSymbol.Show'}
    {attribute 'OPC.UA.DA' := '1'}
    {attribute 'OPC.UA.DA.Access' := '1'}
    actPos : AngularPosition;  (* The actual position (same as parts.physicalAxis!) *)
    {attribute 'TcHmiSymbol.Show'}
    {attribute 'OPC.UA.DA' := '1'}
    {attribute 'OPC.UA.DA.Access' := '1'}
    actVelo : AngularVelocity;  (* The actual velocity (same as parts.physicalAxis!) *)
    {attribute 'TcHmiSymbol.Show'}
    {attribute 'OPC.UA.DA' := '1'}
    {attribute 'OPC.UA.DA.Access' := '1'}
    actAcc : AngularAcceleration;  (* The actual acceleration (same as parts.physicalAxis!) *)
    {attribute 'TcHmiSymbol.Show'}
    {attribute 'OPC.UA.DA' := '1'}
    {attribute 'OPC.UA.DA.Access' := '1'}
    actTorque : Torque;  (* The actual torque on the telescope axis by the ELE motor *)
    {attribute 'TcHmiSymbol.Show'}
    {attribute 'OPC.UA.DA' := '1'}
    {attribute 'OPC.UA.DA.Access' := '1'}
    lida1Position : AngularPosition;  (* Position of the telescope according to LIDA encoder no. 1 *)
    {attribute 'TcHmiSymbol.Show'}
    {attribute 'OPC.UA.DA' := '1'}
    {attribute 'OPC.UA.DA.Access' := '1'}
    lida2Position : AngularPosition;  (* Position of the telescope according to LIDA encoder no. 2 *)
    {attribute 'TcHmiSymbol.Show'}
    {attribute 'OPC.UA.DA' := '1'}
    {attribute 'OPC.UA.DA.Access' := '1'}
    lidaAveragePosition : AngularPosition;  (* Position of the telescope according to the average of the LIDA encoders *)
    {attribute 'TcHmiSymbol.Show'}
    {attribute 'OPC.UA.DA' := '1'}
    {attribute 'OPC.UA.DA.Access' := '1'}
    absoluteEncoderPosition : AngularPosition;  (* Position of the telescope according to the absolute encoder *)
    {attribute 'TcHmiSymbol.Show'}
    statuses : AxesElevationAxisStatuses;  (* Statuses of the state machine *)
    {attribute 'TcHmiSymbol.Show'}
    parts : AxesElevationAxisParts;  (* Parts of the state machine *)
    {attribute 'TcHmiSymbol.Show'}
    processes : AxesElevationAxisProcesses;  (* Processes of the state machine *)
  END_VAR
  VAR_IN_OUT
    {attribute 'TcHmiSymbol.Show'}
    {attribute 'OPC.UA.DA' := '0'}
    {attribute 'TcHmiSymbol.Hide'}
    config : AxesElevationConfig;  (* Reference to the elevation config *)
    {attribute 'TcHmiSymbol.Show'}
    {attribute 'OPC.UA.DA' := '0'}
    {attribute 'TcHmiSymbol.Hide'}
    driveChannel : AX52XXDriveChannel;  (* Reference to the ELE drive channel *)
    {attribute 'TcHmiSymbol.Show'}
    {attribute 'OPC.UA.DA' := '0'}
    {attribute 'TcHmiSymbol.Hide'}
    mainDriveChannel : AX52XXDriveChannel;  (* Reference to the main drive channel (channel A) of the drive *)
  END_VAR

            parts.virtualAxis( isEnabled := isEnabled );
parts.physicalAxis( isEnabled := isEnabled );
parts.lida1( isEnabled := isEnabled );
parts.lida2( isEnabled := isEnabled );
parts.absoluteEncoder();
statuses.busyStatus( isBusy := driveChannel.statuses.busyStatus.busy OR (parts.virtualAxis.statuses.busyStatus.busy OR (parts.physicalAxis.statuses.busyStatus.busy OR (parts.lida1.statuses.busyStatus.busy OR (parts.lida2.statuses.busyStatus.busy OR (processes.moveAbsolute.statuses.busyStatus.busy OR (processes.moveRelative.statuses.busyStatus.busy OR (processes.moveVelocity.statuses.busyStatus.busy OR (processes.reset.statuses.busyStatus.busy OR (processes.moveOutOfLimitSwitch.statuses.busyStatus.busy OR (processes.powerOn.statuses.busyStatus.busy OR (processes.powerOff.statuses.busyStatus.busy OR (processes.doHoming.statuses.busyStatus.busy OR (processes.stop.statuses.busyStatus.busy OR (processes.quickStop.statuses.busyStatus.busy OR (processes.unlockBrake.statuses.busyStatus.busy OR processes.setPosition.statuses.busyStatus.busy))))))))))))))) );
statuses.healthStatus(
    isGood := (driveChannel.statuses.healthStatus.isGood AND (parts.virtualAxis.statuses.healthStatus.isGood AND (parts.physicalAxis.statuses.healthStatus.isGood AND (parts.lida1.statuses.healthStatus.isGood AND (parts.lida2.statuses.healthStatus.isGood AND (parts.absoluteEncoder.statuses.healthStatus.isGood AND (processes.moveAbsolute.statuses.healthStatus.isGood AND (processes.moveRelative.statuses.healthStatus.isGood AND (processes.moveVelocity.statuses.healthStatus.isGood AND (processes.reset.statuses.healthStatus.isGood AND (processes.moveOutOfLimitSwitch.statuses.healthStatus.isGood AND (processes.powerOn.statuses.healthStatus.isGood AND (processes.powerOff.statuses.healthStatus.isGood AND (processes.doHoming.statuses.healthStatus.isGood AND (processes.stop.statuses.healthStatus.isGood AND (processes.quickStop.statuses.healthStatus.isGood AND (processes.unlockBrake.statuses.healthStatus.isGood AND processes.setPosition.statuses.healthStatus.isGood))))))))))))))))) AND ((NOT(slipError)) AND ((NOT(positiveLimitSwitchError)) AND (NOT(negativeLimitSwitchError)))),
    hasWarning := driveChannel.statuses.healthStatus.hasWarning OR (parts.virtualAxis.statuses.healthStatus.hasWarning OR (parts.physicalAxis.statuses.healthStatus.hasWarning OR (parts.lida1.statuses.healthStatus.hasWarning OR (parts.lida2.statuses.healthStatus.hasWarning OR (parts.absoluteEncoder.statuses.healthStatus.hasWarning OR (processes.moveAbsolute.statuses.healthStatus.hasWarning OR (processes.moveRelative.statuses.healthStatus.hasWarning OR (processes.moveVelocity.statuses.healthStatus.hasWarning OR (processes.reset.statuses.healthStatus.hasWarning OR (processes.moveOutOfLimitSwitch.statuses.healthStatus.hasWarning OR (processes.powerOn.statuses.healthStatus.hasWarning OR (processes.powerOff.statuses.healthStatus.hasWarning OR (processes.doHoming.statuses.healthStatus.hasWarning OR (processes.stop.statuses.healthStatus.hasWarning OR (processes.quickStop.statuses.healthStatus.hasWarning OR (processes.unlockBrake.statuses.healthStatus.hasWarning OR processes.setPosition.statuses.healthStatus.hasWarning)))))))))))))))));
statuses.poweredStatus( isEnabled := parts.virtualAxis.statuses.poweredStatus.enabled AND parts.physicalAxis.statuses.poweredStatus.enabled );
processes.moveAbsolute( isEnabled := isEnabled );
processes.moveRelative( isEnabled := isEnabled );
processes.moveVelocity( isEnabled := isEnabled );
processes.reset( isEnabled := isEnabled );
processes.moveOutOfLimitSwitch( isEnabled := isEnabled );
processes.powerOn( isEnabled := isEnabled );
processes.powerOff( isEnabled := isEnabled );
processes.doHoming( isEnabled := isEnabled );
processes.stop( isEnabled := isEnabled );
processes.quickStop( isEnabled := isEnabled );
processes.setPosition( isEnabled := isEnabled );
processes.unlockBrake();

          

{attribute 'TcRpcEnable' := '1'}
METHOD moveAbsolute : RequestResults
  VAR_INPUT
    {attribute 'TcHmiSymbol.Show'}
    units : AxesMoveUnits;
    {attribute 'TcHmiSymbol.Show'}
    value : LREAL;
    {attribute 'TcHmiSymbol.Show'}
    offset : LREAL;
  END_VAR
                  moveAbsolute := THIS^.processes.moveAbsolute.request(
    units := units,
    value := value,
    offset := offset);

                
END_METHOD

{attribute 'TcRpcEnable' := '1'}
METHOD moveRelative : RequestResults
  VAR_INPUT
    {attribute 'TcHmiSymbol.Show'}
    units : AxesMoveUnits;
    {attribute 'TcHmiSymbol.Show'}
    value : LREAL;
  END_VAR
                  moveRelative := THIS^.processes.moveRelative.request(
    units := units,
    value := value);

                
END_METHOD

{attribute 'TcRpcEnable' := '1'}
METHOD moveVelocity : RequestResults
  VAR_INPUT
    {attribute 'TcHmiSymbol.Show'}
    units : AxesMoveVelocityUnits;
    {attribute 'TcHmiSymbol.Show'}
    value : LREAL;
  END_VAR
                  moveVelocity := THIS^.processes.moveVelocity.request(
    units := units,
    value := value);

                
END_METHOD

{attribute 'TcRpcEnable' := '1'}
METHOD reset : RequestResults
                  reset := THIS^.processes.reset.request();

                
END_METHOD

{attribute 'TcRpcEnable' := '1'}
METHOD moveOutOfLimitSwitch : RequestResults
  VAR_INPUT
    {attribute 'TcHmiSymbol.Show'}
    switch : LimitSwitches;
  END_VAR
                  moveOutOfLimitSwitch := THIS^.processes.moveOutOfLimitSwitch.request( switch := switch );

                
END_METHOD

{attribute 'TcRpcEnable' := '1'}
METHOD powerOn : RequestResults
                  powerOn := THIS^.processes.powerOn.request();

                
END_METHOD

{attribute 'TcRpcEnable' := '1'}
METHOD powerOff : RequestResults
                  powerOff := THIS^.processes.powerOff.request();

                
END_METHOD

{attribute 'TcRpcEnable' := '1'}
METHOD doHoming : RequestResults
                  doHoming := THIS^.processes.doHoming.request();

                
END_METHOD

{attribute 'TcRpcEnable' := '1'}
METHOD stop : RequestResults
                  stop := THIS^.processes.stop.request();

                
END_METHOD

{attribute 'TcRpcEnable' := '1'}
METHOD quickStop : RequestResults
                  quickStop := THIS^.processes.quickStop.request();

                
END_METHOD

{attribute 'TcRpcEnable' := '1'}
METHOD setPosition : RequestResults
  VAR_INPUT
    {attribute 'TcHmiSymbol.Show'}
    value : LREAL;
  END_VAR
                  setPosition := THIS^.processes.setPosition.request( value := value );

                
END_METHOD

{attribute 'TcRpcEnable' := '1'}
METHOD unlockBrake : RequestResults
  VAR_INPUT
    {attribute 'TcHmiSymbol.Show'}
    seconds : LREAL;
  END_VAR
                  unlockBrake := THIS^.processes.unlockBrake.request( seconds := seconds );

                
END_METHOD

METHOD _log : BOOL
  VAR_INPUT
    {attribute 'TcHmiSymbol.Show'}
    name : STRING;  (* Name of this function block instance *)
  END_VAR
  VAR_IN_OUT
    {attribute 'TcHmiSymbol.Show'}
    buffer : LogBuffer;  (* Buffer to write all logging to *)
  END_VAR
  VAR
    {attribute 'TcHmiSymbol.Show'}
    subBuffer : LogBuffer;  (* Temporary buffer to write logging by parts (sub-statemachines) to *)
  END_VAR
                  THIS^.parts.virtualAxis._log(
    name := 'virtualAxis',
    buffer := subBuffer);
THIS^.parts.physicalAxis._log(
    name := 'physicalAxis',
    buffer := subBuffer);
THIS^.parts.lida1._log(
    name := 'lida1',
    buffer := subBuffer);
THIS^.parts.lida2._log(
    name := 'lida2',
    buffer := subBuffer);
THIS^.parts.absoluteEncoder._log(
    name := 'absoluteEncoder',
    buffer := subBuffer);
THIS^.processes.moveAbsolute._log(
    name := 'processes.moveAbsolute',
    buffer := subBuffer);
THIS^.processes.moveRelative._log(
    name := 'processes.moveRelative',
    buffer := subBuffer);
THIS^.processes.moveVelocity._log(
    name := 'processes.moveVelocity',
    buffer := subBuffer);
THIS^.processes.reset._log(
    name := 'processes.reset',
    buffer := subBuffer);
THIS^.processes.moveOutOfLimitSwitch._log(
    name := 'processes.moveOutOfLimitSwitch',
    buffer := subBuffer);
THIS^.processes.powerOn._log(
    name := 'processes.powerOn',
    buffer := subBuffer);
THIS^.processes.powerOff._log(
    name := 'processes.powerOff',
    buffer := subBuffer);
THIS^.processes.doHoming._log(
    name := 'processes.doHoming',
    buffer := subBuffer);
THIS^.processes.stop._log(
    name := 'processes.stop',
    buffer := subBuffer);
THIS^.processes.quickStop._log(
    name := 'processes.quickStop',
    buffer := subBuffer);
THIS^.processes.setPosition._log(
    name := 'processes.setPosition',
    buffer := subBuffer);
THIS^.processes.unlockBrake._log(
    name := 'processes.unlockBrake',
    buffer := subBuffer);
LOGGER(
    name := name,
    actualStatus := THIS^.actualStatus,
    previousStatus := THIS^.previousStatus,
    buffer := buffer,
    subBuffer := subBuffer,
    pHealthStatus := ADR(THIS^.statuses.healthStatus),
    pBusyStatus := ADR(THIS^.statuses.busyStatus));

                
END_METHOD
END_FUNCTION_BLOCK

FUNCTION_BLOCK SM_AxesRotationAxis
  VAR_INPUT
    {attribute 'TcHmiSymbol.Show'}
    {attribute 'OPC.UA.DA' := '1'}
    {attribute 'OPC.UA.DA.Access' := '1'}
    id : AxesIds;  (* Id of this axis *)
    {attribute 'TcHmiSymbol.Show'}
    {attribute 'OPC.UA.DA' := '0'}
    {attribute 'TcHmiSymbol.Hide'}
    isEnabled : BOOL;  (* Is control enabled? *)
  END_VAR
  VAR_OUTPUT
    {attribute 'OPC.UA.DA' := '1'}
    {attribute 'OPC.UA.DA.Access' := '1'}
    {attribute 'TcHmiSymbol.Show'}
    actualStatus : STRING;  (* Current status description *)
    {attribute 'TcHmiSymbol.Show'}
    previousStatus : STRING;  (* Previous status description *)
    {attribute 'TcHmiSymbol.Show'}
    {attribute 'OPC.UA.DA' := '1'}
    {attribute 'OPC.UA.DA.Access' := '1'}
    positiveLimitSwitchError : BOOL;  (* TRUE if the positive limit switch has detected the axis *)
    {attribute 'TcHmiSymbol.Show'}
    {attribute 'OPC.UA.DA' := '1'}
    {attribute 'OPC.UA.DA.Access' := '1'}
    negativeLimitSwitchError : BOOL;  (* TRUE if the negative limit switch has detected the axis *)
    {attribute 'TcHmiSymbol.Show'}
    {attribute 'OPC.UA.DA' := '1'}
    {attribute 'OPC.UA.DA.Access' := '1'}
    setPosLimitReached : BOOL;  (* TRUE if the setpoint position has reached its limit *)
    {attribute 'TcHmiSymbol.Show'}
    {attribute 'OPC.UA.DA' := '1'}
    {attribute 'OPC.UA.DA.Access' := '1'}
    deviation1SecAverage : AngularPosition;  (* The deviation between target position and actual position, as a 1 second moving average *)
    {attribute 'TcHmiSymbol.Show'}
    {attribute 'OPC.UA.DA' := '1'}
    {attribute 'OPC.UA.DA.Access' := '1'}
    deviation1SecRMS : AngularPosition;  (* The deviation between target position and actual position, as a 1 second moving RMS error *)
    {attribute 'TcHmiSymbol.Show'}
    {attribute 'OPC.UA.DA' := '1'}
    {attribute 'OPC.UA.DA.Access' := '1'}
    targetPos : AngularPosition;  (* The target position *)
    {attribute 'TcHmiSymbol.Show'}
    {attribute 'OPC.UA.DA' := '1'}
    {attribute 'OPC.UA.DA.Access' := '1'}
    targetOffset : AngularPosition;  (* Cumulative offset of targetPos. Equals targetPos - targetStart *)
    {attribute 'TcHmiSymbol.Show'}
    {attribute 'OPC.UA.DA' := '1'}
    {attribute 'OPC.UA.DA.Access' := '1'}
    targetStart : AngularPosition;  (* Last absolute movement end position of the axis *)
    {attribute 'TcHmiSymbol.Show'}
    {attribute 'OPC.UA.DA' := '1'}
    {attribute 'OPC.UA.DA.Access' := '1'}
    setPos : AngularPosition;  (* The setpoint position (same as parts.physicalAxis!) *)
    {attribute 'TcHmiSymbol.Show'}
    {attribute 'OPC.UA.DA' := '1'}
    {attribute 'OPC.UA.DA.Access' := '1'}
    setVelo : AngularVelocity;  (* The setpoint velocity (same as parts.physicalAxis!) *)
    {attribute 'TcHmiSymbol.Show'}
    {attribute 'OPC.UA.DA' := '1'}
    {attribute 'OPC.UA.DA.Access' := '1'}
    setAcc : AngularAcceleration;  (* The setpoint acceleration (same as parts.physicalAxis!) *)
    {attribute 'TcHmiSymbol.Show'}
    {attribute 'OPC.UA.DA' := '1'}
    {attribute 'OPC.UA.DA.Access' := '1'}
    actPos : AngularPosition;  (* The actual position (same as parts.eleAxis!) *)
    {attribute 'TcHmiSymbol.Show'}
    {attribute 'OPC.UA.DA' := '1'}
    {attribute 'OPC.UA.DA.Access' := '1'}
    actVelo : AngularVelocity;  (* The actual velocity (same as parts.eleAxis!) *)
    {attribute 'TcHmiSymbol.Show'}
    {attribute 'OPC.UA.DA' := '1'}
    {attribute 'OPC.UA.DA.Access' := '1'}
    actAcc : AngularAcceleration;  (* The actual acceleration (same as parts.eleAxis!) *)
    {attribute 'TcHmiSymbol.Show'}
    {attribute 'OPC.UA.DA' := '1'}
    {attribute 'OPC.UA.DA.Access' := '1'}
    actTorque : Torque;  (* The actual torque on the telescope axis by the ELE motor *)
    {attribute 'TcHmiSymbol.Show'}
    statuses : AxesRotationAxisStatuses;  (* Statuses of the state machine *)
    {attribute 'TcHmiSymbol.Show'}
    parts : AxesRotationAxisParts;  (* Parts of the state machine *)
    {attribute 'TcHmiSymbol.Show'}
    processes : AxesRotationAxisProcesses;  (* Processes of the state machine *)
  END_VAR
  VAR_IN_OUT
    {attribute 'TcHmiSymbol.Show'}
    {attribute 'OPC.UA.DA' := '0'}
    {attribute 'TcHmiSymbol.Hide'}
    config : AxesRotationConfig;  (* Reference to the rotation config *)
    {attribute 'TcHmiSymbol.Show'}
    {attribute 'OPC.UA.DA' := '0'}
    {attribute 'TcHmiSymbol.Hide'}
    driveChannel : AX52XXDriveChannel;  (* Reference to the axis drive channel *)
    {attribute 'TcHmiSymbol.Show'}
    {attribute 'OPC.UA.DA' := '0'}
    {attribute 'TcHmiSymbol.Hide'}
    mainDriveChannel : AX52XXDriveChannel;  (* Reference to the main drive channel (channel A) of the drive *)
  END_VAR

            parts.virtualAxis( isEnabled := isEnabled );
parts.physicalAxis( isEnabled := isEnabled );
statuses.busyStatus( isBusy := driveChannel.statuses.busyStatus.busy OR (parts.virtualAxis.statuses.busyStatus.busy OR (parts.physicalAxis.statuses.busyStatus.busy OR (processes.moveAbsolute.statuses.busyStatus.busy OR (processes.moveRelative.statuses.busyStatus.busy OR (processes.moveVelocity.statuses.busyStatus.busy OR (processes.reset.statuses.busyStatus.busy OR (processes.moveOutOfLimitSwitch.statuses.busyStatus.busy OR (processes.powerOn.statuses.busyStatus.busy OR (processes.powerOff.statuses.busyStatus.busy OR (processes.stop.statuses.busyStatus.busy OR (processes.quickStop.statuses.busyStatus.busy OR processes.setPosition.statuses.busyStatus.busy))))))))))) );
statuses.healthStatus(
    isGood := (driveChannel.statuses.healthStatus.isGood AND (parts.virtualAxis.statuses.healthStatus.isGood AND (parts.physicalAxis.statuses.healthStatus.isGood AND (processes.moveAbsolute.statuses.healthStatus.isGood AND (processes.moveRelative.statuses.healthStatus.isGood AND (processes.moveVelocity.statuses.healthStatus.isGood AND (processes.reset.statuses.healthStatus.isGood AND (processes.moveOutOfLimitSwitch.statuses.healthStatus.isGood AND (processes.powerOn.statuses.healthStatus.isGood AND (processes.powerOff.statuses.healthStatus.isGood AND (processes.stop.statuses.healthStatus.isGood AND (processes.quickStop.statuses.healthStatus.isGood AND processes.setPosition.statuses.healthStatus.isGood)))))))))))) AND ((NOT(positiveLimitSwitchError)) AND (NOT(negativeLimitSwitchError))),
    hasWarning := driveChannel.statuses.healthStatus.hasWarning OR (parts.virtualAxis.statuses.healthStatus.hasWarning OR (parts.physicalAxis.statuses.healthStatus.hasWarning OR (processes.moveAbsolute.statuses.healthStatus.hasWarning OR (processes.moveRelative.statuses.healthStatus.hasWarning OR (processes.moveVelocity.statuses.healthStatus.hasWarning OR (processes.reset.statuses.healthStatus.hasWarning OR (processes.moveOutOfLimitSwitch.statuses.healthStatus.hasWarning OR (processes.powerOn.statuses.healthStatus.hasWarning OR (processes.powerOff.statuses.healthStatus.hasWarning OR (processes.stop.statuses.healthStatus.hasWarning OR (processes.quickStop.statuses.healthStatus.hasWarning OR processes.setPosition.statuses.healthStatus.hasWarning))))))))))));
statuses.poweredStatus( isEnabled := parts.virtualAxis.statuses.poweredStatus.enabled AND parts.physicalAxis.statuses.poweredStatus.enabled );
processes.moveAbsolute( isEnabled := isEnabled );
processes.moveRelative( isEnabled := isEnabled );
processes.moveVelocity( isEnabled := isEnabled );
processes.reset( isEnabled := isEnabled );
processes.moveOutOfLimitSwitch( isEnabled := isEnabled );
processes.powerOn( isEnabled := isEnabled );
processes.powerOff( isEnabled := isEnabled );
processes.stop( isEnabled := isEnabled );
processes.quickStop( isEnabled := isEnabled );
processes.setPosition( isEnabled := isEnabled );

          

{attribute 'TcRpcEnable' := '1'}
METHOD moveAbsolute : RequestResults
  VAR_INPUT
    {attribute 'TcHmiSymbol.Show'}
    units : AxesMoveUnits;
    {attribute 'TcHmiSymbol.Show'}
    value : LREAL;
    {attribute 'TcHmiSymbol.Show'}
    offset : LREAL;
  END_VAR
                  moveAbsolute := THIS^.processes.moveAbsolute.request(
    units := units,
    value := value,
    offset := offset);

                
END_METHOD

{attribute 'TcRpcEnable' := '1'}
METHOD moveRelative : RequestResults
  VAR_INPUT
    {attribute 'TcHmiSymbol.Show'}
    units : AxesMoveUnits;
    {attribute 'TcHmiSymbol.Show'}
    value : LREAL;
  END_VAR
                  moveRelative := THIS^.processes.moveRelative.request(
    units := units,
    value := value);

                
END_METHOD

{attribute 'TcRpcEnable' := '1'}
METHOD moveVelocity : RequestResults
  VAR_INPUT
    {attribute 'TcHmiSymbol.Show'}
    units : AxesMoveVelocityUnits;
    {attribute 'TcHmiSymbol.Show'}
    value : LREAL;
  END_VAR
                  moveVelocity := THIS^.processes.moveVelocity.request(
    units := units,
    value := value);

                
END_METHOD

{attribute 'TcRpcEnable' := '1'}
METHOD reset : RequestResults
                  reset := THIS^.processes.reset.request();

                
END_METHOD

{attribute 'TcRpcEnable' := '1'}
METHOD moveOutOfLimitSwitch : RequestResults
  VAR_INPUT
    {attribute 'TcHmiSymbol.Show'}
    switch : LimitSwitches;
  END_VAR
                  moveOutOfLimitSwitch := THIS^.processes.moveOutOfLimitSwitch.request( switch := switch );

                
END_METHOD

{attribute 'TcRpcEnable' := '1'}
METHOD powerOn : RequestResults
                  powerOn := THIS^.processes.powerOn.request();

                
END_METHOD

{attribute 'TcRpcEnable' := '1'}
METHOD powerOff : RequestResults
                  powerOff := THIS^.processes.powerOff.request();

                
END_METHOD

{attribute 'TcRpcEnable' := '1'}
METHOD stop : RequestResults
                  stop := THIS^.processes.stop.request();

                
END_METHOD

{attribute 'TcRpcEnable' := '1'}
METHOD quickStop : RequestResults
                  quickStop := THIS^.processes.quickStop.request();

                
END_METHOD

{attribute 'TcRpcEnable' := '1'}
METHOD setPosition : RequestResults
  VAR_INPUT
    {attribute 'TcHmiSymbol.Show'}
    value : LREAL;
  END_VAR
                  setPosition := THIS^.processes.setPosition.request( value := value );

                
END_METHOD

METHOD _log : BOOL
  VAR_INPUT
    {attribute 'TcHmiSymbol.Show'}
    name : STRING;  (* Name of this function block instance *)
  END_VAR
  VAR_IN_OUT
    {attribute 'TcHmiSymbol.Show'}
    buffer : LogBuffer;  (* Buffer to write all logging to *)
  END_VAR
  VAR
    {attribute 'TcHmiSymbol.Show'}
    subBuffer : LogBuffer;  (* Temporary buffer to write logging by parts (sub-statemachines) to *)
  END_VAR
                  THIS^.parts.virtualAxis._log(
    name := 'virtualAxis',
    buffer := subBuffer);
THIS^.parts.physicalAxis._log(
    name := 'physicalAxis',
    buffer := subBuffer);
THIS^.processes.moveAbsolute._log(
    name := 'processes.moveAbsolute',
    buffer := subBuffer);
THIS^.processes.moveRelative._log(
    name := 'processes.moveRelative',
    buffer := subBuffer);
THIS^.processes.moveVelocity._log(
    name := 'processes.moveVelocity',
    buffer := subBuffer);
THIS^.processes.reset._log(
    name := 'processes.reset',
    buffer := subBuffer);
THIS^.processes.moveOutOfLimitSwitch._log(
    name := 'processes.moveOutOfLimitSwitch',
    buffer := subBuffer);
THIS^.processes.powerOn._log(
    name := 'processes.powerOn',
    buffer := subBuffer);
THIS^.processes.powerOff._log(
    name := 'processes.powerOff',
    buffer := subBuffer);
THIS^.processes.stop._log(
    name := 'processes.stop',
    buffer := subBuffer);
THIS^.processes.quickStop._log(
    name := 'processes.quickStop',
    buffer := subBuffer);
THIS^.processes.setPosition._log(
    name := 'processes.setPosition',
    buffer := subBuffer);
LOGGER(
    name := name,
    actualStatus := THIS^.actualStatus,
    previousStatus := THIS^.previousStatus,
    buffer := buffer,
    subBuffer := subBuffer,
    pHealthStatus := ADR(THIS^.statuses.healthStatus),
    pBusyStatus := ADR(THIS^.statuses.busyStatus));

                
END_METHOD
END_FUNCTION_BLOCK

FUNCTION_BLOCK SM_AxesPointingModelSetup
  VAR_INPUT
    {attribute 'TcHmiSymbol.Show'}
    {attribute 'OPC.UA.DA' := '1'}
    {attribute 'OPC.UA.DA.Access' := '1'}
    editableConfig : AxesPointingModelConfig;  (* Editable configuration of the particular TPOINT model *)
    {attribute 'TcHmiSymbol.Show'}
    {attribute 'OPC.UA.DA' := '0'}
    {attribute 'TcHmiSymbol.Hide'}
    isEnabled : BOOL;  (* Is control enabled? *)
  END_VAR
  VAR_OUTPUT
    {attribute 'OPC.UA.DA' := '1'}
    {attribute 'OPC.UA.DA.Access' := '1'}
    {attribute 'TcHmiSymbol.Show'}
    actualStatus : STRING;  (* Current status description *)
    {attribute 'TcHmiSymbol.Show'}
    previousStatus : STRING;  (* Previous status description *)
    {attribute 'TcHmiSymbol.Show'}
    {attribute 'OPC.UA.DA' := '1'}
    {attribute 'OPC.UA.DA.Access' := '1'}
    config : AxesPointingModelConfig;  (* Active configuration of the particular TPOINT model *)
    {attribute 'TcHmiSymbol.Show'}
    parts : AxesPointingModelSetupParts;  (* Parts of the state machine *)
  END_VAR

            parts.configManager( isEnabled := isEnabled );

          

METHOD _log : BOOL
  VAR_INPUT
    {attribute 'TcHmiSymbol.Show'}
    name : STRING;  (* Name of this function block instance *)
  END_VAR
  VAR_IN_OUT
    {attribute 'TcHmiSymbol.Show'}
    buffer : LogBuffer;  (* Buffer to write all logging to *)
  END_VAR
  VAR
    {attribute 'TcHmiSymbol.Show'}
    subBuffer : LogBuffer;  (* Temporary buffer to write logging by parts (sub-statemachines) to *)
  END_VAR
                  THIS^.parts.configManager._log(
    name := 'configManager',
    buffer := subBuffer);
LOGGER(
    name := name,
    actualStatus := THIS^.actualStatus,
    previousStatus := THIS^.previousStatus,
    buffer := buffer,
    subBuffer := subBuffer);

                
END_METHOD
END_FUNCTION_BLOCK

FUNCTION_BLOCK SM_AxesPointingModelsSetup
  VAR_INPUT
    {attribute 'TcHmiSymbol.Show'}
    {attribute 'OPC.UA.DA' := '0'}
    {attribute 'TcHmiSymbol.Hide'}
    isEnabled : BOOL;  (* Is control enabled? *)
  END_VAR
  VAR_OUTPUT
    {attribute 'OPC.UA.DA' := '1'}
    {attribute 'OPC.UA.DA.Access' := '1'}
    {attribute 'TcHmiSymbol.Show'}
    actualStatus : STRING;  (* Current status description *)
    {attribute 'TcHmiSymbol.Show'}
    previousStatus : STRING;  (* Previous status description *)
    {attribute 'TcHmiSymbol.Show'}
    statuses : AxesPointingModelsSetupStatuses;  (* Statuses of the state machine *)
    {attribute 'TcHmiSymbol.Show'}
    parts : AxesPointingModelsSetupParts;  (* Parts of the state machine *)
  END_VAR

            parts.model0( isEnabled := isEnabled );
parts.model1( isEnabled := isEnabled );
parts.model2( isEnabled := isEnabled );
parts.model3( isEnabled := isEnabled );
parts.model4( isEnabled := isEnabled );
parts.model5( isEnabled := isEnabled );
parts.model6( isEnabled := isEnabled );
parts.model7( isEnabled := isEnabled );
parts.model8( isEnabled := isEnabled );
parts.model9( isEnabled := isEnabled );
statuses.busyStatus( isBusy := parts.model0.parts.configManager.statuses.busyStatus.busy OR (parts.model1.parts.configManager.statuses.busyStatus.busy OR (parts.model2.parts.configManager.statuses.busyStatus.busy OR (parts.model3.parts.configManager.statuses.busyStatus.busy OR (parts.model4.parts.configManager.statuses.busyStatus.busy OR (parts.model5.parts.configManager.statuses.busyStatus.busy OR (parts.model6.parts.configManager.statuses.busyStatus.busy OR (parts.model7.parts.configManager.statuses.busyStatus.busy OR (parts.model8.parts.configManager.statuses.busyStatus.busy OR parts.model9.parts.configManager.statuses.busyStatus.busy)))))))) );
statuses.healthStatus(
    isGood := parts.model0.parts.configManager.statuses.healthStatus.isGood AND (parts.model1.parts.configManager.statuses.healthStatus.isGood AND (parts.model2.parts.configManager.statuses.healthStatus.isGood AND (parts.model3.parts.configManager.statuses.healthStatus.isGood AND (parts.model4.parts.configManager.statuses.healthStatus.isGood AND (parts.model5.parts.configManager.statuses.healthStatus.isGood AND (parts.model6.parts.configManager.statuses.healthStatus.isGood AND (parts.model7.parts.configManager.statuses.healthStatus.isGood AND (parts.model8.parts.configManager.statuses.healthStatus.isGood AND parts.model9.parts.configManager.statuses.healthStatus.isGood)))))))),
    hasWarning := parts.model0.parts.configManager.statuses.healthStatus.hasWarning OR (parts.model1.parts.configManager.statuses.healthStatus.hasWarning OR (parts.model2.parts.configManager.statuses.healthStatus.hasWarning OR (parts.model3.parts.configManager.statuses.healthStatus.hasWarning OR (parts.model4.parts.configManager.statuses.healthStatus.hasWarning OR (parts.model5.parts.configManager.statuses.healthStatus.hasWarning OR (parts.model6.parts.configManager.statuses.healthStatus.hasWarning OR (parts.model7.parts.configManager.statuses.healthStatus.hasWarning OR (parts.model8.parts.configManager.statuses.healthStatus.hasWarning OR parts.model9.parts.configManager.statuses.healthStatus.hasWarning)))))))));

          

METHOD _log : BOOL
  VAR_INPUT
    {attribute 'TcHmiSymbol.Show'}
    name : STRING;  (* Name of this function block instance *)
  END_VAR
  VAR_IN_OUT
    {attribute 'TcHmiSymbol.Show'}
    buffer : LogBuffer;  (* Buffer to write all logging to *)
  END_VAR
  VAR
    {attribute 'TcHmiSymbol.Show'}
    subBuffer : LogBuffer;  (* Temporary buffer to write logging by parts (sub-statemachines) to *)
  END_VAR
                  THIS^.parts.model0._log(
    name := 'model0',
    buffer := subBuffer);
THIS^.parts.model1._log(
    name := 'model1',
    buffer := subBuffer);
THIS^.parts.model2._log(
    name := 'model2',
    buffer := subBuffer);
THIS^.parts.model3._log(
    name := 'model3',
    buffer := subBuffer);
THIS^.parts.model4._log(
    name := 'model4',
    buffer := subBuffer);
THIS^.parts.model5._log(
    name := 'model5',
    buffer := subBuffer);
THIS^.parts.model6._log(
    name := 'model6',
    buffer := subBuffer);
THIS^.parts.model7._log(
    name := 'model7',
    buffer := subBuffer);
THIS^.parts.model8._log(
    name := 'model8',
    buffer := subBuffer);
THIS^.parts.model9._log(
    name := 'model9',
    buffer := subBuffer);
LOGGER(
    name := name,
    actualStatus := THIS^.actualStatus,
    previousStatus := THIS^.previousStatus,
    buffer := buffer,
    subBuffer := subBuffer,
    pHealthStatus := ADR(THIS^.statuses.healthStatus),
    pBusyStatus := ADR(THIS^.statuses.busyStatus));

                
END_METHOD
END_FUNCTION_BLOCK

FUNCTION_BLOCK SM_AxesIO
  VAR_INPUT
    {attribute 'TcHmiSymbol.Show'}
    {attribute 'OPC.UA.DA' := '1'}
    {attribute 'OPC.UA.DA.Access' := '1'}
    isEnabled : BOOL;  (* Is control enabled? *)
  END_VAR
  VAR_OUTPUT
    {attribute 'OPC.UA.DA' := '1'}
    {attribute 'OPC.UA.DA.Access' := '1'}
    {attribute 'TcHmiSymbol.Show'}
    actualStatus : STRING;  (* Current status description *)
    {attribute 'TcHmiSymbol.Show'}
    previousStatus : STRING;  (* Previous status description *)
    {attribute 'TcHmiSymbol.Show'}
    statuses : AxesIOStatuses;  (* Statuses of the state machine *)
    {attribute 'TcHmiSymbol.Show'}
    parts : AxesIOParts;  (* Parts of the state machine *)
  END_VAR

            parts.aziDrive( isEnabled := isEnabled );
parts.ablDrive( isEnabled := isEnabled );
parts.eleDrive( isEnabled := isEnabled );
parts.TA_AZID(
    id := 'TA:AZID',
    typeId := 'AX5206');
parts.TA_ABLD(
    id := 'TA:ABLD',
    typeId := 'AX5206');
parts.TA_ELED(
    id := 'TA:ELED',
    typeId := 'AX5206');
parts.TE_COU(
    id := 'TE:COU',
    typeId := 'EK1100');
parts.TE_EN1(
    id := 'TE:EN1',
    typeId := 'EL5101');
parts.TE_EN2(
    id := 'TE:EN2',
    typeId := 'EL5101');
parts.TE_EN3(
    id := 'TE:EN3',
    typeId := 'EL5101');
parts.TE_EN4(
    id := 'TE:EN4',
    typeId := 'EL5101');
parts.TE_EN5(
    id := 'TE:EN5',
    typeId := 'EL5101');
parts.TE_EN6(
    id := 'TE:EN6',
    typeId := 'EL5101');
parts.TE_EN7(
    id := 'TE:EN7',
    typeId := 'EL5002');
statuses.healthStatus( isGood := parts.aziDrive.statuses.healthStatus.isGood AND (parts.ablDrive.statuses.healthStatus.isGood AND (parts.eleDrive.statuses.healthStatus.isGood AND (parts.TA_AZID.statuses.healthStatus.isGood AND (parts.TA_ABLD.statuses.healthStatus.isGood AND (parts.TA_ELED.statuses.healthStatus.isGood AND (parts.TE_COU.statuses.healthStatus.isGood AND (parts.TE_EN1.statuses.healthStatus.isGood AND (parts.TE_EN1.statuses.healthStatus.isGood AND (parts.TE_EN2.statuses.healthStatus.isGood AND (parts.TE_EN3.statuses.healthStatus.isGood AND (parts.TE_EN4.statuses.healthStatus.isGood AND (parts.TE_EN5.statuses.healthStatus.isGood AND (parts.TE_EN6.statuses.healthStatus.isGood AND parts.TE_EN7.statuses.healthStatus.isGood))))))))))))) );

          

METHOD _log : BOOL
  VAR_INPUT
    {attribute 'TcHmiSymbol.Show'}
    name : STRING;  (* Name of this function block instance *)
  END_VAR
  VAR_IN_OUT
    {attribute 'TcHmiSymbol.Show'}
    buffer : LogBuffer;  (* Buffer to write all logging to *)
  END_VAR
  VAR
    {attribute 'TcHmiSymbol.Show'}
    subBuffer : LogBuffer;  (* Temporary buffer to write logging by parts (sub-statemachines) to *)
  END_VAR
                  THIS^.parts.aziDrive._log(
    name := 'aziDrive',
    buffer := subBuffer);
THIS^.parts.ablDrive._log(
    name := 'ablDrive',
    buffer := subBuffer);
THIS^.parts.eleDrive._log(
    name := 'eleDrive',
    buffer := subBuffer);
THIS^.parts.TA_AZID._log(
    name := 'TA_AZID',
    buffer := subBuffer);
THIS^.parts.TA_ABLD._log(
    name := 'TA_ABLD',
    buffer := subBuffer);
THIS^.parts.TA_ELED._log(
    name := 'TA_ELED',
    buffer := subBuffer);
THIS^.parts.TE_COU._log(
    name := 'TE_COU',
    buffer := subBuffer);
THIS^.parts.TE_EN1._log(
    name := 'TE_EN1',
    buffer := subBuffer);
THIS^.parts.TE_EN2._log(
    name := 'TE_EN2',
    buffer := subBuffer);
THIS^.parts.TE_EN3._log(
    name := 'TE_EN3',
    buffer := subBuffer);
THIS^.parts.TE_EN4._log(
    name := 'TE_EN4',
    buffer := subBuffer);
THIS^.parts.TE_EN5._log(
    name := 'TE_EN5',
    buffer := subBuffer);
THIS^.parts.TE_EN6._log(
    name := 'TE_EN6',
    buffer := subBuffer);
THIS^.parts.TE_EN7._log(
    name := 'TE_EN7',
    buffer := subBuffer);
LOGGER(
    name := name,
    actualStatus := THIS^.actualStatus,
    previousStatus := THIS^.previousStatus,
    buffer := buffer,
    subBuffer := subBuffer,
    pHealthStatus := ADR(THIS^.statuses.healthStatus));

                
END_METHOD
END_FUNCTION_BLOCK

FUNCTION_BLOCK AxesSetTargetProcess EXTENDS BaseProcess
  VAR_INPUT
    {attribute 'OPC.UA.DA' := '1'}
    {attribute 'TcHmiSymbol.Show'}
    set : AxesSetTargetProcessArgs;  (* Arguments to be set, before writing do_request TRUE *)
  END_VAR
  VAR_OUTPUT
    {attribute 'OPC.UA.DA' := '1'}
    {attribute 'OPC.UA.DA.Access' := '1'}
    {attribute 'TcHmiSymbol.Show'}
    get : AxesSetTargetProcessArgs;  (* Arguments in use by the process, if do_request was accepted *)
  END_VAR

            IF do_request THEN
    do_request_result := request(
    alphaUnits := set.alphaUnits,
    alpha := set.alpha,
    deltaUnits := set.deltaUnits,
    delta := set.delta,
    muUnits := set.muUnits,
    muAlpha := set.muAlpha,
    muDelta := set.muDelta,
    parallax := set.parallax,
    radialVelocity := set.radialVelocity,
    epoch := set.epoch);
    do_request := FALSE;
END_IF;
SUPER^();

          

